# B&R Automation Studio project NAELD004C00R10L518F00 (part 36)

#### Act_Background.st
```iecst
(** 2020-05-26 **)
ACTION Act_Background:

	//Update Parameter
	IF bModuleOK = TRUE THEN

		tyParamInMove.diPosInUM		:= p_diMovePosInUM;
		tyParamInMove.diDistInUM	:= p_diMoveDistInUM;
		tyParamInMove.diVelInUMPS	:= p_diMoveVelInUMPS;
		tyParamInMove.diAcc			:= p_diMoveAcc;
		tyParamInMove.diDec			:= p_diMoveDec;

		fMotionCANUpdtDat(ADR(tyParamOut) , p_tyParamInConvert , tyParamOutDriver , tyParamInDriver , tyParamInMove , p_tyParamInHm , p_bDir, p_eNtParamMotorType);

		bWidthPosDiff	:= (tyParamOut.bIsHomed = FALSE) OR ((ABS((fAWWidthToPosInUM(p_diGoWidth , p_diWidthAtHmPos)) - tyParamOut.diActualPosInUM)) > 500);

		//p_tyParamInConvert.diPitchInUM	:= fPitchCalc(p_diWidthOffsetInUM , p_diMaxWidthInUM , p_diMinWidthInUM , p_diPitchInUM);

		fbFullMovAbsBl.tyParamInConvert					:= p_tyParamInConvert;

		IF p_bDir = TRUE THEN
			bOpenSen	:= tyParamOut.bFwdLmtSen;
			bCloseSen	:= tyParamOut.bRevLmtSen;
		ELSE
			bOpenSen	:= tyParamOut.bRevLmtSen;
			bCloseSen	:= tyParamOut.bFwdLmtSen;
		END_IF

		CASE p_eNtParamMotorType OF
			DeltaAsdaA2:
				CASE tyParamOut.udiAxisErrID OF
					8976:	sAxisErrTxt	:= 'Over Current';
					12560:	sAxisErrTxt	:= 'Over Voltage';
					12576:	sAxisErrTxt	:= 'Under Voltage';
					12592:	sAxisErrTxt	:= 'Input Power Phase Loss';
					12816:	sAxisErrTxt	:= 'Regeneration Error';
					12848:	sAxisErrTxt	:= 'Overload';
					12849:	sAxisErrTxt	:= 'Pre-overload Warning';
					13056:	sAxisErrTxt	:= 'U,V,W Wiring Error';
					16912:	sAxisErrTxt	:= 'IGBT Temperature Error';
					21296:	sAxisErrTxt	:= 'Memory Error';
					21569:	sAxisErrTxt	:= 'Emergency Stop Activated';
					21570:	sAxisErrTxt	:= 'Forward Limit Switch Error';
					21571:	sAxisErrTxt	:= 'Reverse Limit Switch Error';
					21572:	sAxisErrTxt	:= 'Forward Software Limit';
					21573:	sAxisErrTxt	:= 'Reverse Software Limit';
					21760:	sAxisErrTxt	:= 'DSP Firmware Upgrade';
					25088:	sAxisErrTxt	:= 'CANopen SYNC Error';
					25360:	sAxisErrTxt	:= 'CANopen Data Initial Error';
					25376:	sAxisErrTxt	:= 'Adjustment Error';
					28961:	sAxisErrTxt	:= 'Motor Protection Error';
					28962:	sAxisErrTxt	:= 'Motor Error';
					29445:	sAxisErrTxt	:= 'Encoder Error';
					29446:	sAxisErrTxt	:= 'Encoder Output Error';
					29968:	sAxisErrTxt	:= 'Serial Communication Error';
					29984:	sAxisErrTxt	:= 'Serial Communication Time Out';
					33024:	sAxisErrTxt	:= 'CANbus Error (Bus-off)';
					33040:	sAxisErrTxt	:= 'CANopen SDO receive buffer overrun';
					33056:	sAxisErrTxt	:= 'CANbus Error (Warning)';
					33072:	sAxisErrTxt	:= 'Node Guarding or Heartbeat Error';
					33280:	sAxisErrTxt	:= 'CANopen PDO Object Error';
					33792:	sAxisErrTxt	:= 'Over Speed';
					34304:	sAxisErrTxt	:= 'Abnormal Pulse Control Command';
					34320:	sAxisErrTxt	:= 'Full Closed Loop Excessive Deviation';
					34321:	sAxisErrTxt	:= 'Excessive Deviation';
				END_CASE

			SchneiderLexium28:
				CASE tyParamOut.udiAxisErrID OF
					8724:	sAxisErrTxt	:= 'Over Current';
					8976:	sAxisErrTxt	:= 'Motor Overload';
					8977:	sAxisErrTxt	:= 'Drive overload (foldback)';
					9088:	sAxisErrTxt	:= 'Calculated offsets for current sensors out OF range';
					9089:	sAxisErrTxt := 'Motor phase missing';
					9090:	sAxisErrTxt := 'Overcurrent detected at one OF the digital outputs';
					12560:	sAxisErrTxt	:= 'DC Bus Over Voltage';
					12576:	sAxisErrTxt	:= 'DC Bus Under Voltage';
					12672:	sAxisErrTxt	:= 'Braking Resistor Overload';
					12673:	sAxisErrTxt	:= 'Safety function Safe Torque Off (STO) triggered';
					12674:	sAxisErrTxt	:= 'DC bus voltage measurement';
					12675:	sAxisErrTxt	:= 'Missing mains supply, undervoltage mains supply';
					12676:	sAxisErrTxt := 'The encoder supply voltage has dropped under operational value';
					12677:	sAxisErrTxt := 'The multi turn encoder battery voltage has dropped under 3 Vdc';
					12678:	sAxisErrTxt := 'Internal position sync error detected.';
					12679:	sAxisErrTxt := 'Generic error code of the multi turn module is detected';
					12697:	sAxisErrTxt := 'Braking resistor overload';
					16512:	sAxisErrTxt	:= 'Drive overtemperature (IPM)';
					16513:	sAxisErrTxt	:= 'Drive overtemperature (controller)';
					16534:	sAxisErrTxt := 'Temperature sensor inoperative';
					17168:	sAxisErrTxt	:= 'Power stage overtemperature';
					17280:	sAxisErrTxt := 'The encoder temperature is too high';
					17424:	sAxisErrTxt	:= 'Motor overtemperature';
					21808:	sAxisErrTxt	:= 'System error detected (nonvolatilememory)';
					21893:	sAxisErrTxt	:= 'Error detected in non-volatile memory';
					21889:	sAxisErrTxt	:= 'System error detected (nonvolatile memory)';
					21890:	sAxisErrTxt	:= 'System error detected (CAN power supply)';
					21891:	sAxisErrTxt	:= 'System error detected (selftest)';
					21894:	sAxisErrTxt	:= 'System error detected (NV ACCESS)';
					25472:	sAxisErrTxt	:= 'Target position rejected';
					25985:	sAxisErrTxt	:= 'System error detected(FPGA)';
					28816:	sAxisErrTxt	:= 'System error detected (FPGA does NOT match firmware)';
					28817:	sAxisErrTxt	:= 'Emergency Stop Activated';
					28961:	sAxisErrTxt := 'Motor blocked';
					29080:	sAxisErrTxt := 'Commutation error detected';
					29568:  sAxisErrTxt	:= 'Error detected in communication with motor encoder';
					29574:	sAxisErrTxt	:= 'Drive is not synchronous wit master cycle';
					29581:	sAxisErrTxt := 'System error detected (encoder)';
					29587:	sAxisErrTxt	:= 'Encoder overvoltage or overcurrent';
					29592:	sAxisErrTxt := 'The returned position value are no longer considered valid';
					29593:	sAxisErrTxt := 'The multi turn encoder requires an explicit configuration command';
					30081:	sAxisErrTxt := 'Target position rejected';
					30082:	sAxisErrTxt := 'No target values received via the fieldbus';
					33072:	sAxisErrTxt	:= 'CANopen: Heartbeat error detected';
					33296:	sAxisErrTxt := 'R_PDO is too short';
					33921:	sAxisErrTxt	:= 'Actual Motor Velocity Too High';
					33553:	sAxisErrTxt	:= 'Motor torque too high FOR an excessive period OF time';
					33664:	sAxisErrTxt := 'Unstable current loop';
					33922:	sAxisErrTxt := 'Velocity deviation too high';
					34321:	sAxisErrTxt	:= 'Position deviation too high';
					34432:	sAxisErrTxt := 'Position deviation via signal output function MC_OK';
					34441:	sAxisErrTxt := 'Position deviation too high (following error)';
					61568:	sAxisErrTxt	:= 'Fieldbus: Communication	error detected';
					65282:	sAxisErrTxt	:= 'Not possible to read data of electronic motor nameplate';
					65296:	sAxisErrTxt	:= 'Forward Limit Switch Error';
					65297:	sAxisErrTxt	:= 'Reverse Limit Switch Error';
					65281:	sAxisErrTxt := 'System error detected';
					65298:	sAxisErrTxt	:= 'Forward Software Limit';
					65299:	sAxisErrTxt	:= 'Reverse Software Limit';
					65301:	sAxisErrTxt := 'The encoder firmware cannot operate on the provided hardware';

				END_CASE

			EstunPronet:
				CASE tyParamOut.udiAxisErrID OF
					65281:	sAxisErrTxt	:= 'Parameter breakdown';//A01
					65282:	sAxisErrTxt	:= 'AD shift channels breakdown';
					65283:	sAxisErrTxt	:= 'Overspeed';
					65284:	sAxisErrTxt	:= 'Overload';
					65285:	sAxisErrTxt := 'Position error counteroverflow ';
					65286:	sAxisErrTxt := 'Position error pulse overflow';
					65287:	sAxisErrTxt	:= 'The setting of electronic gear or given pulse frequency is not reasonable';
					65288:	sAxisErrTxt	:= 'The 1st channel of current detection is wrong.';
					65289:	sAxisErrTxt	:= 'The 2nd channel of current detection is wrong.';
					65290:	sAxisErrTxt	:= 'Incremental Encoder is break off.';//A10
					65292:	sAxisErrTxt	:= 'Overcurrent';
					65293:	sAxisErrTxt	:= 'Overvoltage';
					65294:	sAxisErrTxt	:= 'Undervoltage';
					65295:	sAxisErrTxt := 'Bleeder resistor error';
					65296:	sAxisErrTxt := 'Regeneration error';
					65297:	sAxisErrTxt := 'Resolver error';
					65298:	sAxisErrTxt := 'IGBT superheat alarm';
					65299:	sAxisErrTxt := 'Motor overheat alarm';
					65300:	sAxisErrTxt := 'Power line phase shortage';//A20
					65301:	sAxisErrTxt	:= 'Instantaneous power off alarm';
					65302:	sAxisErrTxt	:= 'Motor temperature detection sensor is break off.';
					65303:	sAxisErrTxt := 'Brake overcurrent alarm';//A23
					65305:	sAxisErrTxt := 'Motor power line U overcurrent';//A25
					65306:	sAxisErrTxt := 'Motor power line V overcurrent';//A26
					65307:	sAxisErrTxt := 'Motor power line W overcurrent';//A27
					65322:	sAxisErrTxt	:= 'Servomotor type error';//A42
					65323:	sAxisErrTxt	:= 'Servo drive type error';
					65325:	sAxisErrTxt	:= 'Absolute encoder multiturn information error';
					65326:	sAxisErrTxt	:= 'Absolute encoder multiturn information overflow';
					65327:	sAxisErrTxt	:= 'Battery voltage below 2.5V';
					65328:	sAxisErrTxt	:= 'Battery voltage below 3.1V';//A48
					65330:	sAxisErrTxt := 'Serial encoder communication overtime ';//A50
					65331:	sAxisErrTxt := 'Absolute encoder overspeed alarm detected';
					65332:  sAxisErrTxt	:= 'Absolute state of serial encoder error';
					65333:	sAxisErrTxt	:= 'Serial encoder calcaution error';
					65334:	sAxisErrTxt := 'Parity bit or end bit in serial encoder control domain error';
					65335:	sAxisErrTxt	:= 'Serial encoder communication data checking error';
					65336:	sAxisErrTxt := 'End bit in serial encoder control domain error';
					65338:	sAxisErrTxt := 'Serial encoder data empty';
					65339:	sAxisErrTxt := 'Serial encoder data format error';
					65340:	sAxisErrTxt := 'Communication module not detected ';//A60
					65341:	sAxisErrTxt := 'Communication unsuccessful';
					65342:	sAxisErrTxt := 'Servo drive can not receive the period data of communication module ';
					65343:	sAxisErrTxt := 'Communication module can not receive the servo drive response data.';
					65344:	sAxisErrTxt := 'Communication module and bus connectionless';
					65346:	sAxisErrTxt := 'CAN communication abnormal';
					65347:	sAxisErrTxt := 'Receiving heartbeat timeout';
					65349:	sAxisErrTxt := 'Synchronization signal monitoring cycle is longer than setting';
					65362: sAxisErrTxt	:= 'Torque output alarm';
				END_CASE
		END_CASE

	ELSE

		tyParamOut.bAxisErr			:= FALSE;
		tyParamOut.bFwdLmtSen		:= FALSE;
		tyParamOut.bInPos			:= FALSE;
		tyParamOut.bIsHomed			:= FALSE;
		tyParamOut.bPosDiff			:= TRUE;
		tyParamOut.bPwrOn			:= FALSE;
		tyParamOut.bRevLmtSen		:= FALSE;
		tyParamOut.bStopped			:= TRUE;
		tyParamOut.diActualPosInUM	:= 0;
		tyParamOut.diHmAcc			:= 0;
		tyParamOut.diHmSpdForSwitch	:= 0;
		tyParamOut.diHmSpdForZero	:= 0;
		tyParamOut.diProfileAcc		:= 0;
		tyParamOut.diProfileDec		:= 0;
		tyParamOut.udiAxisErrID		:= 0;

		bWidthPosDiff				:= TRUE;

	END_IF

	//Abnormal Movement
//	IF eStatus1 <> Error THEN
//		IF p_bOps = TRUE AND eStatus = Idle THEN
//			IF (ABS(tyParamOut.diActualPosInUM - diActualPosInUMOld) > 2000) AND (ABS(tyParamOut.diActualPosInUM - diActualPosInUMOld) < 10000) THEN
//				eStatus1	:= Error;
//				udiStatus1	:= 10000;	//Axis Move Abnormally By External Force
//
//				fMotionCANRstCtrlWord(ADR(tyParamOutDriver));
//				p_eAct	:= PPActIdle;
//				eStat	:= PPActIdle;
//			END_IF
//		ELSE
//			diActualPosInUMOld	:= tyParamOut.diActualPosInUM;
//		END_IF
//	END_IF

	//Reset Error
	IF (eStatus1 = Error) AND bRstErr THEN
		eStatus1	:= Idle;
		udiStatus1	:= 0;
	END_IF

	//Request Position To Movement Out Of Range
	IF p_bOps
		AND((tyParamInMove.diPosInUM < p_diMinAbsPosInUM) OR (tyParamInMove.diPosInUM > p_diMaxAbsPosInUM))
		AND (eStatus2 <> Error) THEN
		eStatus2	:= Error;
		udiStatus2	:= 10029;	//Request Absolute Position Out Of Range

		fMotionCANRstCtrlWord(ADR(tyParamOutDriver));
		p_eAct	:= PPActIdle;
		eStat	:= PPActIdle;
	END_IF

	//Reset Error
	IF (eStatus2 = Error) AND bRstErr THEN
		eStatus2	:= Idle;
		udiStatus2	:= 0;
	END_IF

	//Sensor Interrupt
	IF (bNotInterruptible = TRUE OR bJogging) AND eStatus3 <> Error THEN

		IF p_bInletSensor = TRUE THEN
			eStatus3	:= Error;
			udiStatus3	:= 10030;	//Inlet Sensor Interrupt Auto Width Movement

			fMotionCANRstCtrlWord(ADR(tyParamOutDriver));
			p_eAct	:= PPActIdle;
			eStat	:= PPActIdle;

		ELSIF p_bOutletSensor = TRUE THEN
			eStatus3	:= Error;
			udiStatus3	:= 10031;	//Outlet Sensor Interrupt Auto Width Movement

			fMotionCANRstCtrlWord(ADR(tyParamOutDriver));
			p_eAct	:= PPActIdle;
			eStat	:= PPActIdle;

		ELSIF p_bClearSensor = TRUE THEN
			eStatus3	:= Error;
			udiStatus3	:= 10032;	//Clear Sensor Interrupt Auto Width Movement

			fMotionCANRstCtrlWord(ADR(tyParamOutDriver));
			p_eAct	:= PPActIdle;
			eStat	:= PPActIdle;

		ELSIF p_bMiddleSensor = TRUE THEN
			eStatus3	:= Error;
			udiStatus3	:= 10033;	//Middle Sensor Interrupt Auto Width Movement

			fMotionCANRstCtrlWord(ADR(tyParamOutDriver));
			p_eAct	:= PPActIdle;
			eStat	:= PPActIdle;

		ELSIF p_bInterruptSensor = TRUE THEN
			eStatus3	:= Error;
			udiStatus3	:= 10034;	//Sensor Interrupt Auto Width Movement

			fMotionCANRstCtrlWord(ADR(tyParamOutDriver));
			p_eAct	:= PPActIdle;
			eStat	:= PPActIdle;

		ELSIF p_bCloseInterruptSensor = TRUE AND bJogOpen = FALSE THEN
			eStatus3	:= Error;
			udiStatus3	:= 10047;	//Sensor Interrupt Auto Width Movement

			fMotionCANRstCtrlWord(ADR(tyParamOutDriver));
			p_eAct	:= PPActIdle;
			eStat	:= PPActIdle;

		ELSIF p_bOpenInterruptSensor = TRUE AND bJogClose = FALSE THEN
			eStatus3	:= Error;
			udiStatus3	:= 10048;	//Sensor Interrupt Auto Width Movement

			fMotionCANRstCtrlWord(ADR(tyParamOutDriver));
			p_eAct	:= PPActIdle;
			eStat	:= PPActIdle;
		END_IF

	END_IF

	//Reset Error
	IF (eStatus3 = Error AND bRstErr)
		OR (p_bOpenInterruptSensor AND eStat = PPActJogClose)
		OR (p_bCloseInterruptSensor AND eStat = PPActJogOpen)
		THEN
		eStatus3	:= Idle;
		udiStatus3	:= 0;
	END_IF

	IF bRstErr THEN
		udiStatus	:= 0;
		bJogging	:= FALSE;
		bJogClose	:= FALSE;
		bJogOpen	:= FALSE;
	END_IF

	fbServoModuleOk(IN:= bModuleOK);
	fbServoModuleNotOk(IN:= bModuleOK = FALSE);
	IF fbServoModuleNotOk.Q AND udiStatus <> 10001 THEN

		bModuleNotOK		:= TRUE;
		bModuleNotOKLock	:= TRUE;
		usiRstStep	:= 0;
		tyParamOutDriver.uiCtrlword_6040	:= 0;
		tyParamOutDriver.siModOfOpt_6060	:= 0;
		tyParamOutDriver.diTargetPos_607A	:= 0;
		tyParamOutDriver.udiMoveSpd_6081	:= 0;
		tyParamOutDriver.siHmMethod_6098	:= 0;
		tyParamOutDriver.diJogVel_60FF		:= 0;

		CASE p_eNtParamMotorType OF

			DeltaAsdaA2:
				fbModuleOK(bModuleOK:= FALSE);
				IF eStatus = Idle THEN
					eAct	:= PPActRstNode;
				END_IF

				IF (eStatus = Done OR eStatus = Error)AND eStat = PPActRstNode THEN

					eAct	:= PPActIdle;
				END_IF

			EstunPronet:
				fbModuleOK(bModuleOK:= FALSE);
				IF eStatus = Idle THEN
					eAct	:= PPActRstNode;
				END_IF

				IF (eStatus = Done OR eStatus = Error)AND eStat = PPActRstNode THEN

					eAct	:= PPActIdle;
				END_IF

			SchneiderLexium28:
			// Do Nothing
		END_CASE

	ELSIF bModuleNotOK = TRUE AND fbServoModuleOk.Q THEN

		CASE usiRstStep OF

			0:
				IF eStatus = Idle THEN
					eAct	:= PPActRstAxisErr;
				END_IF

				IF eStatus = Done AND eStat = PPActRstAxisErr THEN
					eAct	:= PPActIdle;
					usiRstStep	:= 4;
				END_IF

			4: tyParamOutDriver.siModOfOpt_6060 := 1;
				usiRstStep	:= 5;

			5: tyParamOutDriver.siModOfOpt_6060 := 1;
				fbRstNodeTimer(IN:=TRUE);

				IF tyParamInDriver.siModOfOptDisp_6061 = 1 THEN
					usiRstStep	:= 6;
					fbRstNodeTimer(IN:=FALSE);
				ELSIF fbRstNodeTimer.Q THEN
					usiRstStep	:= 8;
					fbRstNodeTimer(IN:=FALSE);
				END_IF

			6: tyParamOutDriver.siModOfOpt_6060 := 6;
				fbRstNodeTimer(IN:=FALSE);
				usiRstStep	:= 7;

			7: tyParamOutDriver.siModOfOpt_6060 := 6;
				fbRstNodeTimer(IN:=TRUE);

				IF tyParamInDriver.siModOfOptDisp_6061 = 6 THEN
					usiRstStep	:= 10;
					fbRstNodeTimer(IN:=FALSE);
				ELSIF fbRstNodeTimer.Q THEN
					usiRstStep	:= 9;
					fbRstNodeTimer(IN:=FALSE);
				END_IF

			8:	fbModuleOK(bEn := TRUE, bModuleOK:= FALSE);
				fbRstNodeTimer(IN:=FALSE);
				usiRstStep	:= 9;

			9:	fbModuleOK(bModuleOK:= FALSE);
				IF eStatus = Idle THEN
					eAct	:=PPActRstNode;
				END_IF

				IF eStatus = Done AND eStat = PPActRstNode THEN
					usiRstStep	:= 0;
					eAct		:= PPActIdle;
				END_IF

			10:IF eStatus = Idle THEN
					eAct	:= PPActRstAxisErr;
				END_IF

				IF eStatus = Done AND eStat = PPActRstAxisErr THEN
					eAct			:=PPActIdle;
					usiRstStep	:= 11;
				END_IF

			11:

				IF eStatus = Idle THEN
					eAct	:= PPActSDOWrite;
				END_IF

				IF eStatus = Done AND eStat = PPActSDOWrite THEN
					eAct			:= PPActIdle;
					usiRstStep	:= 13;

				ELSIF udiStatus = 10028 THEN
					eAct			:= PPActIdle;
					usiRstStep	:= 13;
				END_IF

			13: bModuleNotOK	:= FALSE;
				usiRstStep	:= 0;
		END_CASE
	ELSE
		eAct	:= PPActIdle;

	END_IF

	IF tyParamOut.bPosDiff = FALSE THEN
		tyParamOutDriver.uiCtrlword_6040.4	:= FALSE;
	END_IF

END_ACTION
```

#### Act_InitGlobal.st
```iecst
(** 2019-04-09 **)
ACTION Act_InitGlobal:

	(* Always Change If Project Change *)

	//Pass Data To Link
	p_bLinkOpsRun ACCESS p_OpsRun;
	p_bLinkStartupRun ACCESS p_StartupRun;
	p_bLinkPullConvPullerExtCtrl ACCESS p_PullConvPullerExtCtrl;
	p_bLinkPullConvPullerRetCtrl ACCESS p_PullConvPullerRetCtrl;
	p_bLinkDIPullerExtRS ACCESS p_DIPullerExtRS;
	p_bLinkDIPullerRetRS ACCESS p_DIPullerRetRS;
	p_bLinkDIPullerExtSlwRS ACCESS p_DIPullerExtSlwSen;
	p_bLinkDIPullerRetSlwRS ACCESS p_DIPullerRetSlwSen;
	p_dintLinkPullerRetSpd ACCESS p_ProdRcpCurrRcp1MtrPshrExtSpd;
	p_dintLinkPullerRetTrq ACCESS p_ProdRcpCurrRcp1MtrPshrExtTorq;
	p_bLinkDIPullerRotHmRS ACCESS p_DIPullerRotHmRS;

	p_diLinkMag1TravPos ACCESS p_MagRcpCurrRcpMag1TravPos;
	p_diLinkMag2TravPos ACCESS p_MagRcpCurrRcpMag2TravPos;
	p_diLinkMag3TravPos ACCESS p_MagRcpCurrRcpMag3TravPos;
	p_diLinkTravActualPos ACCESS p_TravActualPos;
	p_bProjCurtainSenPrep ACCESS p_NtParamProjCurtainSenPrep; //shutter become individual : interrupt sensor
	p_diRcp1MtrPshrExtTorq ACCESS p_ProdRcpCurrRcp1MtrPshrExtTorq;
	p_bMagWidthChkSen ACCESS p_DIMagWidthChkSen;
	p_tyLinkTorqParam ACCESS p_NtParamPPTorqParam;

	//Pass Data To Internal Use
	p_udiRstErr ACCESS p_RstErrReset;
	p_bEn ACCESS p_DISimServoEn;
	p_bPrep ACCESS p_NtParamProjServoPullPusherPrep;
	p_bOps ACCESS p_OpsStatusRun;
	p_bManual ACCESS p_UIMnlMod;
	p_tyTuning ACCESS p_NtParamPPTuning;
//	p_diJogVelInUMPS ACCESS p_UIMnlPPJogSpd;
	p_diMovePosInUM ACCESS p_UIMnlPPTargetPos;
	p_diMoveDistInUM ACCESS p_UIMnlPPStepSize;
	p_diMoveVelInUMPS ACCESS p_NtParamPPAutoSpd;
	p_diMoveAcc ACCESS p_NtParamPPAcc;
	p_diMoveDec ACCESS p_NtParamPPDec;
	p_diWidthOffsetInUM ACCESS p_NtParamWidthOffset;
	p_bDir ACCESS p_NtParamPPDir;
	p_bDirBl ACCESS p_NtParamPPDirBl;
	p_usiNode ACCESS p_NtParamPPNode;
	p_sDevice ACCESS p_NtParamPPDevice;
	p_sProgNm ACCESS p_NtParamPPProgNm;
	p_diMoveBacklashDistInUM ACCESS p_NtParamPPMovBlDistInUM;
	p_diPitchInUM ACCESS p_NtParamPPPitchInUM;
	p_tyParamInHm ACCESS p_NtParamPPParamInHm;
	p_tyParamInConvert ACCESS p_NtParamPPParamInConvert;
	p_bNtSettingsLoadDone ACCESS p_StartupNtSettingsLoadDone;
	p_eNtParamMotorType ACCESS p_NtParamPPMotorType;

	p_bInletShutterCloseRS ACCESS p_DIInShutterCloseRS;
	p_bOutletShutterCloseRS ACCESS p_DIOutShutterCloseRS;
	p_bProjInletShutPrep ACCESS p_NtParamProjInletShutPrep;
	p_bProjOutletShutPrep ACCESS p_NtParamProjOutletShutPrep;

	p_bInletShutterCloseRS2 ACCESS p_DIInShutterCloseRS2;
	p_bInletShutterCloseRS3 ACCESS p_DIInShutterCloseRS3;

	(* Always Change If Project Change *)

END_ACTION
```

#### Act_Initial.st
```iecst
(** 2020-03-16 **)
ACTION Act_Initial:

	//Initial
	sStatTxt	:= a_sStatText[eStat];

	tyParamInMove.diBacklashDistInUM	:= p_diMoveBacklashDistInUM;
	tyParamInMove.diAcc					:= p_diMoveAcc;
	tyParamInMove.diDec					:= p_diMoveDec;

	//p_tyParamInConvert.diPitchInUM	:= fPitchCalc(p_diWidthOffsetInUM , p_diMaxWidthInUM , p_diMinWidthInUM , p_diPitchInUM);

	fbModuleOK.sDevice	:= p_sDevice;
	fbModuleOK.usiNode	:= p_usiNode;
	fbModuleOK.tDlyTm	:= T#5s;
	fbModuleOK(bEn := FALSE);

	fbSDOWrite.sDevice	:= p_sDevice;
	fbSDOWrite.usiNode	:= p_usiNode;
	fbSDOWrite.eMotorType	:= p_eNtParamMotorType;
	fbSDOWrite(bEn := FALSE);

	fbFullMovAbsBl.p_tyParamOutDriver				:= ADR(tyParamOutDriver);
	fbFullMovAbsBl.tyParamInMove.diBacklashDistInUM	:= p_diMoveBacklashDistInUM;
	fbFullMovAbsBl.tyParamInMove.diAcc				:= p_diMoveAcc;
	fbFullMovAbsBl.tyParamInMove.diDec				:= p_diMoveDec;
	//fbFullMovAbsBl.tyParamInConvert					:= p_tyParamInConvert;
	fbFullMovAbsBl.bDir								:= p_bDir;
	fbFullMovAbsBl.bDirBl							:= p_bDirBl;
	fbFullMovAbsBl.bNoIndexPulse					:= p_bNoIndexPulse;
	fbFullMovAbsBl.eMotorType						:= p_eNtParamMotorType;
	fbFullMovAbsBl(bEn := FALSE);

	fbFullMovAbs.p_tyParamOutDriver					:= ADR(tyParamOutDriver);
	fbFullMovAbs.tyParamInMove.diBacklashDistInUM	:= p_diMoveBacklashDistInUM;
	fbFullMovAbs.tyParamInMove.diAcc				:= p_diMoveAcc;
	fbFullMovAbs.tyParamInMove.diDec				:= p_diMoveDec;
	fbFullMovAbs.tyParamInConvert					:= p_tyParamInConvert;
	fbFullMovAbs.bDir								:= p_bDir;
	fbFullMovAbs.bNoIndexPulse						:= p_bNoIndexPulse;
	fbFullMovAbs.eMotorType							:= p_eNtParamMotorType;
	fbFullMovAbs(bEn := FALSE);

	fbFullHm.p_tyParamOutDriver	:= ADR(tyParamOutDriver);
	fbFullHm.bDir				:= p_bDir;
	fbFullHm.bNoIndexPulse		:= p_bNoIndexPulse;
	fbFullHm.eMotorType			:= p_eNtParamMotorType;
	fbFullHm(bEn := FALSE);

	fbPwrOn.p_tyParamOutDriver	:= ADR(tyParamOutDriver);
	fbPwrOn.eMotorType			:= p_eNtParamMotorType;
	fbPwrOn(bEn := FALSE);

	fbPwrOff.p_tyParamOutDriver	:= ADR(tyParamOutDriver);
	fbPwrOff.eMotorType			:= p_eNtParamMotorType;
	fbPwrOff(bEn := FALSE);

	fbHoming.p_tyParamOutDriver	:= ADR(tyParamOutDriver);
	fbHoming.bDir				:= p_bDir;
	fbHoming.bNoIndexPulse		:= p_bNoIndexPulse;
	fbHoming.eMotorType			:= p_eNtParamMotorType;
	fbHoming(bEn := FALSE);

	fbMovAbs.p_tyParamOutDriver					:= ADR(tyParamOutDriver);
	fbMovAbs.tyParamInMove.diBacklashDistInUM	:= p_diMoveBacklashDistInUM;
	fbMovAbs.tyParamInMove.diAcc				:= p_diMoveAcc;
	fbMovAbs.tyParamInMove.diDec				:= p_diMoveDec;
	fbMovAbs.tyParamInConvert					:= p_tyParamInConvert;
	fbMovAbs.bDir								:= p_bDir;
	fbMovAbs.eMotorType							:= p_eNtParamMotorType;
	fbMovAbs(bEn := FALSE);

	fbMovRel.p_tyParamOutDriver					:= ADR(tyParamOutDriver);
	fbMovRel.tyParamInMove.diBacklashDistInUM	:= p_diMoveBacklashDistInUM;
	fbMovRel.tyParamInMove.diAcc				:= p_diMoveAcc;
	fbMovRel.tyParamInMove.diDec				:= p_diMoveDec;
	fbMovRel.tyParamInConvert					:= p_tyParamInConvert;
	fbMovRel.bDir								:= p_bDir;
	fbMovRel.eMotorType							:= p_eNtParamMotorType;
	fbMovRel(bEn := FALSE);

	fbJog.p_tyParamOutDriver	:= ADR(tyParamOutDriver);
	fbJog.tyParamInConvert		:= p_tyParamInConvert;
	fbJog.eMotorType			:= p_eNtParamMotorType;
	fbJog(bEn := FALSE);

	fbRstAxisErr.p_tyParamOutDriver	:= ADR(tyParamOutDriver);
	fbRstAxisErr(bEn := FALSE);

	fbStop.p_tyParamOutDriver	:= ADR(tyParamOutDriver);
	fbStop(bEn := FALSE);

	fbSDOWriteTorque.pDevice := ADR(p_sDevice);
	fbSDOWriteTorque.node	 := p_usiNode;

	fbSDOWriteTorque.index	:= 16#210C;
	fbSDOWriteTorque.subindex	:= 0;
	fbSDOWriteTorque.datalen	:= 2;

	bModuleNotOK	:= TRUE;

END_ACTION
```

#### Act_InitLocal.st
```iecst
(** 2020-05-26 **)
ACTION Act_InitLocal:

	//Input Reference Link To Local Variable
	p_eAct ACCESS ADR(eAct);
	p_udiRstErr ACCESS ADR(udiRstErr);
	p_bPrep ACCESS ADR(bPrep);
	p_bEn ACCESS ADR(bEn);
	p_bDis ACCESS ADR(bDis);
	p_bOps ACCESS ADR(bOps);
	p_bManual ACCESS ADR(bManual);
	p_diWidthAtHmPos ACCESS ADR(diWidthAtHmPos);
	p_tyTuning ACCESS ADR(tyTuning);
	p_diGoWidth ACCESS ADR(diGoWidth);
	p_diJogVelInUMPS ACCESS ADR(diJogVelInUMPS);
	p_diMovePosInUM ACCESS ADR(diMovePosInUM);
	p_diMoveDistInUM ACCESS ADR(diMoveDistInUM);
	p_diMoveVelInUMPS ACCESS ADR(diMoveVelInUMPS);
	p_diMoveAcc ACCESS ADR(diMoveAcc);
	p_diMoveDec ACCESS ADR(diMoveDec);
	p_diMinAbsPosInUM ACCESS ADR(diMinAbsPosInUM);
	p_diMaxAbsPosInUM ACCESS ADR(diMaxAbsPosInUM);
	p_diMinWidthInUM ACCESS ADR(diMinWidthInUM);
	p_diMaxWidthInUM ACCESS ADR(diMaxWidthInUM);
	p_diWidthOffsetInUM ACCESS ADR(diWidthOffsetInUM);
	p_bInletSensor ACCESS ADR(bInletSensor);
	p_bOutletSensor ACCESS ADR(bOutletSensor);
	p_bClearSensor ACCESS ADR(bClearSensor);
	p_bMiddleSensor ACCESS ADR(bMiddleSensor);
	p_bInterruptSensor ACCESS ADR(bInterruptSensor);
	p_bOpenInterruptSensor ACCESS ADR(bOpenInterruptSensor);
	p_bCloseInterruptSensor ACCESS ADR(bCloseInterruptSensor);
	p_bDir ACCESS ADR(bDir);
	p_bDirBl ACCESS ADR(bDirBl);
	p_bNoIndexPulse ACCESS ADR(bNoIndexPulse);
	p_usiNode ACCESS ADR(usiNode);
	p_sDevice ACCESS ADR(sDevice);
	p_sProgNm ACCESS ADR(sProgNm);
	p_diMoveBacklashDistInUM ACCESS ADR(diMoveBacklashDistInUM);
	p_diPitchInUM ACCESS ADR(diPitchInUM);
	p_tyParamInHm ACCESS ADR(tyParamInHm);
	p_tyParamInConvert ACCESS ADR(tyParamInConvert);
	p_bNtSettingsLoadDone ACCESS ADR(bNtSettingsLoadDone);
	p_eNtParamMotorType ACCESS ADR(eMotorType);
	p_diServoTorque ACCESS ADR(diServoTorque);
	p_diRcp1MtrPshrExtTorq ACCESS ADR(diRcp1MtrPshrExtTorq);
END_ACTION
```

#### Act_Link.st
```iecst
(** 2019-03-29 **)
ACTION Act_Link:
	diRcp1MtrPshrExtTorq	 := p_tyLinkTorqParam.usiStartTorque + (((p_diRcp1MtrPshrExtTorq -10)/10)*p_tyLinkTorqParam.uiRatio/100);//15~30N , Rcp1 torque

	IF p_bProjInletShutPrep = TRUE THEN

		IF p_bProjCurtainSenPrep = FALSE THEN //standard
			IF p_bInletShutterCloseRS
				THEN
				bInterruptSensor1 := TRUE;
			ELSE
				bInterruptSensor1 := FALSE;
			END_IF
		ELSE
			IF eStat <> PPActJogClose THEN
				IF ABS(p_diLinkMag1TravPos - p_diLinkTravActualPos) < 500 THEN
					bInterruptSensor1 := p_bInletShutterCloseRS;
				ELSIF ABS(p_diLinkMag2TravPos - p_diLinkTravActualPos) < 500 THEN
					bInterruptSensor1 := p_bInletShutterCloseRS2;
				ELSIF ABS(p_diLinkMag3TravPos - p_diLinkTravActualPos) < 500 THEN
					bInterruptSensor1 := p_bInletShutterCloseRS3;
				END_IF
			END_IF
		END_IF
	ELSE
		bInterruptSensor1 := FALSE;
	END_IF

//	IF p_bProjOutletShutPrep = TRUE THEN
//		IF p_bOutletShutterCloseRS
//			THEN
//			bInterruptSensor2 := TRUE;
//		ELSE
//			bInterruptSensor2 := FALSE;
//		END_IF
//	ELSE
//		bInterruptSensor2 := FALSE;
//	END_IF

//	IF (usiJogFwdStep = 40 AND p_eAct = PPActJogOpen) OR (usiJogRevStep = 40 AND p_eAct = PPActJogClose) THEN
//		bInterruptSensor3	:= NOT p_bMagWidthChkSen;
//	END_IF
//	IF p_eAct = PPActIdle OR p_eAct = PPActStop THEN
//		bInterruptSensor3  := FALSE;
//	END_IF

	p_bInterruptSensor := bInterruptSensor3 OR bInterruptSensor2 OR bInterruptSensor1;// OR p_bLinkSafetyRelay = FALSE;

END_ACTION
```

#### Act_LinkAction.st
```iecst
(** 2019-10-21 **)
ACTION Act_LinkAction:

	IF bModuleNotOK THEN
		p_eAct ACCESS ADR(eAct);
	ELSE
		IF p_bLinkStartupRun = TRUE THEN
			p_eAct ACCESS p_StartupServoPPAct;
		ELSIF p_bLinkOpsRun = TRUE OR p_bManual = TRUE THEN
			IF p_bLinkPullConvPullerExtCtrl AND NOT bJogFwdDone
				//AND NOT p_bLinkDIPullerExtRS
				THEN
				bJogStopDone := FALSE;

				CASE usiJogFwdStep OF

					0:
						memcpy(ADR(fbSDOWriteTorque.data0),ADR(udiMaxTorque),1);
						memcpy(ADR(fbSDOWriteTorque.data1),ADR(udiMaxTorque)+1,1);
						IF eStat <> PPActIdle THEN
							p_eAct := PPActIdle;
							usiJogFwdStep := 20;
						ELSE
							usiJogFwdStep := 20;
						END_IF

					20:
						fbSDOWriteTorque(enable := TRUE);
						IF fbSDOWriteTorque.status = 65535 THEN
							usiJogFwdStep := 22;
						END_IF

					22:
						fbSDOWriteTorque(enable := TRUE);
						IF fbSDOWriteTorque.status = 0 THEN
							fbSDOWriteTorque(enable := FALSE);
							usiJogFwdStep := 30;
						END_IF

					30:
						IF tyParamOut.bPwrOn = FALSE THEN
							p_eAct := PPActPwrOn;

							IF tyParamOut.bPwrOn THEN
								p_eAct := PPActIdle;
								usiJogFwdStep := 40;
							END_IF
						ELSE
							p_eAct := PPActIdle;
							usiJogFwdStep := 40;

						END_IF

					40:
						p_eAct := PPActJogOpen;

						IF EDGEPOS(p_bLinkDIPullerExtSlwRS) THEN
							bExtSlowSpd := TRUE;
							p_eAct := PPActIdle;
						END_IF

						IF p_bLinkDIPullerExtSlwRS OR p_bLinkDIPullerExtRS  THEN
							p_diJogVelInUMPS := diSlowSpeed;

						ELSE
							IF p_bManual THEN
								p_diJogVelInUMPS ACCESS p_UIMnlPPJogSpd;
							ELSE
									p_diJogVelInUMPS := udiJogSpdAuto; //325000;//290000;
							END_IF
						END_IF

					//	IF (eStat = PPActJogOpen AND eMainStatus = Done)
					//		OR p_bLinkDIPullerExtRS
						IF p_bLinkDIPullerExtRS
							THEN
							p_eAct := PPActIdle;
							p_diJogVelInUMPS := 0;
							usiJogFwdStep := 50;

						END_IF

					50:
						p_eAct := PPActJogStop;
						p_diJogVelInUMPS := 0;
						IF (eStat = PPActJogStop AND eMainStatus = Done)
							THEN
							p_eAct := PPActIdle;
							usiJogFwdStep := 0;
							bJogFwdDone := TRUE;
						END_IF

				END_CASE

			ELSIF p_bLinkPullConvPullerRetCtrl AND NOT bJogRevDone
				//AND NOT p_bLinkDIPullerRetRS
				THEN
				bJogStopDone := FALSE;
				CASE usiJogRevStep OF

					0:
						IF p_bManual THEN
							memcpy(ADR(fbSDOWriteTorque.data0),p_UIMnlMtrPshrRetTorq,1);
							memcpy(ADR(fbSDOWriteTorque.data1),p_UIMnlMtrPshrRetTorq+1,1);
						ELSE
							memcpy(ADR(fbSDOWriteTorque.data0),ADR(diRcp1MtrPshrExtTorq),1);
							memcpy(ADR(fbSDOWriteTorque.data1),ADR(diRcp1MtrPshrExtTorq)+1,1);
						END_IF
						IF eStat <> PPActIdle THEN
							p_eAct := PPActIdle;
							usiJogRevStep := 20;
						ELSE
							usiJogRevStep := 20;
						END_IF

					20:
						fbSDOWriteTorque(enable := TRUE);
						IF fbSDOWriteTorque.status = 65535 THEN
							usiJogRevStep := 22;
						END_IF

					22:
						fbSDOWriteTorque(enable := TRUE);
						IF fbSDOWriteTorque.status = 0 THEN
							fbSDOWriteTorque(enable := FALSE);
							usiJogRevStep := 30;
						END_IF

					30:
						IF tyParamOut.bPwrOn = FALSE THEN
							p_eAct := PPActPwrOn;
							IF tyParamOut.bPwrOn THEN
								p_eAct := PPActIdle;
								usiJogRevStep := 40;
							END_IF
						ELSE
							p_eAct := PPActIdle;
							usiJogRevStep := 40;

						END_IF

					40:
						p_eAct := PPActJogClose;

						IF EDGEPOS(p_bLinkDIPullerRetSlwRS) THEN
							p_eAct := PPActIdle;
						END_IF

						IF p_bLinkDIPullerRetSlwRS OR p_bLinkDIPullerRetRS THEN
							p_diJogVelInUMPS := diSlowSpeed;
						ELSE
							IF p_bManual THEN
								p_diJogVelInUMPS ACCESS p_UIMnlPPJogSpd;
							ELSE
								p_diJogVelInUMPS := p_dintLinkPullerRetSpd * uiJogSpdRatio; //40625//36250
							END_IF

						END_IF

					//	IF (eStat = PPActJogClose AND eMainStatus = Done)
					//		OR p_bLinkDIPullerRetRS
						IF p_bLinkDIPullerRetRS
							THEN
							p_eAct := PPActIdle;
							p_diJogVelInUMPS := 0;
							usiJogRevStep := 50;

						END_IF

					50:
						p_eAct := PPActJogStop;
						p_diJogVelInUMPS := 0;
						IF (eStat = PPActJogStop AND eMainStatus = Done)
						THEN
							p_eAct := PPActIdle;
							usiJogRevStep := 0;
							bJogRevDone := TRUE;
						END_IF

				END_CASE
			ELSE

				IF bJogStopDone = FALSE THEN
					p_eAct := PPActJogStop;
				END_IF

				usiJogFwdStep := 0;
				usiJogRevStep := 0;
				p_diJogVelInUMPS := 0;

				IF eStat = PPActJogStop AND eMainStatus = Done THEN
					p_eAct := PPActIdle;
					bJogStopDone := TRUE;
				END_IF

				IF tyParamInDriver.uiErrCode_603F <> 0 THEN //error 12592
					tyParamOutDriver.uiCtrlword_6040 := 0; //0111 (7)> 1111 (15)
				END_IF

			END_IF

		ELSE
			IF bRstAndExt = FALSE THEN
				p_eAct ACCESS ADR(eAct);
				usiJogFwdStep := 0;
				usiJogRevStep := 0;
				usiRstJogStep := 0;
				p_diJogVelInUMPS := 0;
				IF bModuleNotOK = FALSE THEN
					IF eStatus <> Idle THEN
						p_eAct := PPActIdle;
						IF eStat = PPActIdle AND eMainStatus = Done THEN
							p_eAct := PPActIdle;
						END_IF
					END_IF
				END_IF
			ELSIF p_bLinkDIPullerRetRS OR p_bLinkDIPullerRotHmRS THEN
				bRstAndExt := FALSE;

			ELSE //reset do extend
				p_eAct ACCESS ADR(eAct);
				CASE usiRstJogStep OF
					0:
						fbPwrOnDlyTmr(IN:=tyParamOut.bPwrOn = FALSE);
						IF tyParamOut.bPwrOn = FALSE AND fbPwrOnDlyTmr.Q THEN
							p_eAct := PPActPwrOn;

							IF tyParamOut.bPwrOn THEN
								fbPwrOnDlyTmr(IN:=FALSE);
								p_eAct := PPActIdle;
								usiRstJogStep := 1;
							END_IF
						ELSE
							fbPwrOnDlyTmr(IN:=FALSE);
							p_eAct := PPActIdle;
							usiRstJogStep := 1;

						END_IF
					1:
						p_eAct := PPActJogOpen;

						IF EDGEPOS(p_bLinkDIPullerExtSlwRS) THEN
							p_eAct := PPActIdle;
						END_IF

						IF p_bLinkDIPullerExtSlwRS OR p_bLinkDIPullerExtRS OR bExtSlowSpd THEN
							p_diJogVelInUMPS := diSlowSpeed;

						ELSE
							p_diJogVelInUMPS := 12000; //50%

						END_IF

						IF p_bLinkDIPullerExtRS	THEN
							p_eAct := PPActIdle;
							p_diJogVelInUMPS := 0;
							usiRstJogStep := 2;
							bTurnToHm	:= TRUE; // output
							bExtSlowSpd := FALSE;

						END_IF

					2:
						p_eAct := PPActJogStop;
						p_diJogVelInUMPS := 0;
						IF (eStat = PPActJogStop AND eMainStatus = Done)
							THEN
							p_eAct := PPActIdle;
							bRstAndExt := FALSE;
						END_IF
				END_CASE

			END_IF
		END_IF //end run/manual
	END_IF

	IF EDGENEG(p_bManual) OR EDGENEG(p_bLinkOpsRun) OR EDGENEG(p_bLinkStartupRun) THEN
		tyParamOutDriver.uiCtrlword_6040	:= 0;
	END_IF

	IF (eStat = PPActJogClose AND p_bLinkDIPullerRetRS)
		OR (eStat = PPActJogOpen AND p_bLinkDIPullerExtRS)
		THEN
		p_diJogVelInUMPS := 0;
	END_IF

	IF p_bLinkDIPullerRetRS = FALSE THEN
		bJogRevDone := FALSE;
	END_IF

	IF p_bLinkDIPullerExtRS = FALSE THEN
		bJogFwdDone := FALSE;
	END_IF

END_ACTION
```

#### Act_Main.st
```iecst
(** 2020-05-26 **)
ACTION Act_Main:

	//Main
IF bModuleNotOK = FALSE THEN

		CASE eStat OF

			PPActIdle:
				IF eStatus <> Idle THEN	//Reset Data
					//Private
					fbStop(bEn := FALSE);
					fbRstAxisErr(bEn := FALSE);
					fbJog(bEn := FALSE);
					fbMovRel(bEn := FALSE);
					fbMovAbs(bEn := FALSE);
					fbHoming(bEn := FALSE);
					fbPwrOff(bEn := FALSE);
					fbPwrOn(bEn := FALSE);
					fbFullHm(bEn := FALSE);
					fbFullMovAbs(bEn := FALSE);
					fbFullMovAbsBl(bEn := FALSE);
					fbSDOWrite(bEn := FALSE);
					fbTm(IN := FALSE);
					usiStep				:= 0;
					usiCount			:= 0;
					bNotInterruptible	:= FALSE;
					tyParamOutDriver.uiCtrlword_6040.7	:= FALSE;
					sStatTxt	:= a_sStatText[eStat];

				END_IF

				eStatus	:= Idle;

				IF EDGENEG(p_bManual) THEN
					fMotionCANRstCtrlWord(ADR(tyParamOutDriver));
				END_IF

			PPActGoWidth:
				IF (eStatus = Idle OR eStatus = Busy) THEN

					eStatus	:= Busy;

					sStatTxt	:= a_sStatText[eStat];

					bNotInterruptible	:= TRUE;

					CASE usiStep OF
						0:	//Wait For Motion Parameter Update
							p_diMovePosInUM	:= fAWWidthToPosInUM(p_diGoWidth , p_diWidthAtHmPos);
							usiStep	:= 1;

						1:	//Check Position Difference
							IF tyParamOut.bPosDiff = TRUE THEN
								usiStep	:= 2;
							ELSE
								eStatus	:= Done;
							END_IF

						2:	//Move
							fbFullMovAbsBl.tyParamInDriver					:= tyParamInDriver;
							fbFullMovAbsBl.tyParamInMove.diPosInUM			:= p_diMovePosInUM;
							fbFullMovAbsBl.tyParamInMove.diDistInUM			:= p_diMoveDistInUM;
							fbFullMovAbsBl.tyParamInMove.diVelInUMPS		:= p_diMoveVelInUMPS;
							fbFullMovAbsBl.tyParamInMove.diAcc				:= p_diMoveAcc;
							fbFullMovAbsBl.tyParamInMove.diDec				:= p_diMoveDec;
							fbFullMovAbsBl.tyParamOut						:= tyParamOut;
							fbFullMovAbsBl(bEn := TRUE);

							IF fbFullMovAbsBl.udiStatus = 0 THEN
								eStatus	:= Done;
							ELSIF fbFullMovAbsBl.udiStatus < 65534 THEN
								eStatus		:= Error;

								IF fbFullMovAbsBl.udiStatus = 1401 THEN
									udiStatus	:= 10002;	//Power On Time Out While Going New Width
								ELSIF fbFullMovAbsBl.udiStatus = 1402 THEN
									udiStatus	:= 10003;	//Homing Time Out While Going New Width
								ELSIF fbFullMovAbsBl.udiStatus = 1403 THEN
									udiStatus	:= 10004;	//Move Absolute Time Out While Going New Width
								ELSIF fbFullMovAbsBl.udiStatus = 1405 THEN
									udiStatus	:= 10005;	//Stop Motion Time Out While Going New Width
								ELSIF fbFullMovAbsBl.udiStatus = 1408 THEN
									udiStatus	:= 10006;	//Axis Error Reset Failed While Going New Width
								ELSIF fbFullMovAbsBl.udiStatus = 1409 THEN
									udiStatus	:= 10007;	//Axis Error Occur In Move Absolute While Going New Width
								ELSIF fbFullMovAbsBl.udiStatus = 1411 THEN
									udiStatus	:= 10008;	//Axis Error Occur In Homing While Going New Width
								ELSIF fbFullMovAbsBl.udiStatus = 1412 THEN
									udiStatus	:= 10009;	//Homing Done But Home Flag Is Not Activated While Going New Width
								ELSIF fbFullMovAbsBl.udiStatus = 1413 THEN
									udiStatus	:= 10010;	//Forward Limit Activated In Homing While Going New Width
								ELSIF fbFullMovAbsBl.udiStatus = 1414 THEN
									udiStatus	:= 10011;	//Reverse Limit Activated In Homing While Going New Width
								ELSIF fbFullMovAbsBl.udiStatus = 1415 THEN
									udiStatus	:= 10012;	//Forward Limit Activated In Move Absolute While Going New Width
								ELSIF fbFullMovAbsBl.udiStatus = 1416 THEN
									udiStatus	:= 10013;	//Reverse Limit Activated In Move Absolute While Going New Width
								ELSE
									udiStatus	:= fbFullMovAbsBl.udiStatus;
								END_IF
							END_IF

					END_CASE

				END_IF

			PPActGoWidthOff:
				IF (eStatus = Idle OR eStatus = Busy) THEN

					eStatus	:= Busy;

					sStatTxt	:= a_sStatText[eStat];

					bNotInterruptible	:= TRUE;

					CASE usiStep OF
						0:	//Wait For Motion Parameter Update
							p_diMovePosInUM	:= fAWWidthToPosInUM(p_diGoWidth , p_diWidthAtHmPos);
							usiStep	:= 1;

						1:	//Check Position Difference
							IF tyParamOut.bPosDiff = TRUE THEN
								usiStep	:= 2;
							ELSE
								eStatus	:= Done;
							END_IF

						2:	//Move
							fbFullMovAbsBl.tyParamInDriver					:= tyParamInDriver;
							fbFullMovAbsBl.tyParamInMove.diPosInUM			:= p_diMovePosInUM;
							fbFullMovAbsBl.tyParamInMove.diDistInUM			:= p_diMoveDistInUM;
							fbFullMovAbsBl.tyParamInMove.diVelInUMPS		:= p_diMoveVelInUMPS;
							fbFullMovAbsBl.tyParamInMove.diAcc				:= p_diMoveAcc;
							fbFullMovAbsBl.tyParamInMove.diDec				:= p_diMoveDec;
							fbFullMovAbsBl.tyParamOut						:= tyParamOut;
							fbFullMovAbsBl(bEn := TRUE);

							IF fbFullMovAbsBl.udiStatus = 0 THEN
								usiStep	:= 3;
							ELSIF fbFullMovAbsBl.udiStatus < 65534 THEN
								eStatus		:= Error;

								IF fbFullMovAbsBl.udiStatus = 1401 THEN
									udiStatus	:= 10035;	//Power On Time Out While Going New Width And Off
								ELSIF fbFullMovAbsBl.udiStatus = 1402 THEN
									udiStatus	:= 10036;	//Homing Time Out While Going New Width And Off
								ELSIF fbFullMovAbsBl.udiStatus = 1403 THEN
									udiStatus	:= 10037;	//Move Absolute Time Out While Going New Width And Off
								ELSIF fbFullMovAbsBl.udiStatus = 1405 THEN
									udiStatus	:= 10038;	//Stop Motion Time Out While Going New Width And Off
								ELSIF fbFullMovAbsBl.udiStatus = 1408 THEN
									udiStatus	:= 10039;	//Axis Error Reset Failed While Going New Width And Off
								ELSIF fbFullMovAbsBl.udiStatus = 1409 THEN
									udiStatus	:= 10040;	//Axis Error Occur In Move Absolute While Going New Width And Off
								ELSIF fbFullMovAbsBl.udiStatus = 1411 THEN
									udiStatus	:= 10041;	//Axis Error Occur In Homing While Going New Width And Off
								ELSIF fbFullMovAbsBl.udiStatus = 1412 THEN
									udiStatus	:= 10042;	//Homing Done But Home Flag Is Not Activated While Going New Width And Off
								ELSIF fbFullMovAbsBl.udiStatus = 1413 THEN
									udiStatus	:= 10043;	//Forward Limit Activated In Homing While Going New Width And Off
								ELSIF fbFullMovAbsBl.udiStatus = 1414 THEN
									udiStatus	:= 10044;	//Reverse Limit Activated In Homing While Going New Width And Off
								ELSIF fbFullMovAbsBl.udiStatus = 1415 THEN
									udiStatus	:= 10045;	//Forward Limit Activated In Move Absolute While Going New Width And Off
								ELSIF fbFullMovAbsBl.udiStatus = 1416 THEN
									udiStatus	:= 10046;	//Reverse Limit Activated In Move Absolute While Going New Width And Off
								ELSE
									udiStatus	:= fbFullMovAbsBl.udiStatus;
								END_IF
							END_IF

						3:	//Turn Off Motor
							fMotionCANRstCtrlWord(ADR(tyParamOutDriver));
							eStatus	:= Done;

					END_CASE

				END_IF

			PPActFullHm:
				IF (eStatus = Idle OR eStatus = Busy) THEN

					eStatus	:= Busy;

					sStatTxt	:= a_sStatText[eStat];

					bNotInterruptible	:= TRUE;

					fbFullHm.tyParamInDriver	:= tyParamInDriver;
					fbFullHm.tyParamOut			:= tyParamOut;
					fbFullHm(bEn := TRUE);

					IF fbFullHm.udiStatus = 0 THEN
						eStatus	:= Done;
					ELSIF fbFullHm.udiStatus < 65534 THEN
						eStatus		:= Error;

						IF fbFullHm.udiStatus = 1401 THEN
							udiStatus	:= 10014;	//Power On Time Out While Full Homing
						ELSIF fbFullHm.udiStatus = 1402 THEN
							udiStatus	:= 10015;	//Homing Time Out While Full Homing
						ELSIF fbFullHm.udiStatus = 1405 THEN
							udiStatus	:= 10016;	//Stop Motion Time Out While Full Homing
						ELSIF fbFullHm.udiStatus = 1408 THEN
							udiStatus	:= 10017;	//Axis Error Reset Failed While Full Homing
						ELSIF fbFullHm.udiStatus = 1411 THEN
							udiStatus	:= 10018;	//Axis Error Occur In Homing While Full Homing
						ELSIF fbFullHm.udiStatus = 1412 THEN
							udiStatus	:= 10019;	//Homing Done But Home Flag Is Not Activated While Full Homing
						ELSIF fbFullHm.udiStatus = 1413 THEN
							udiStatus	:= 10020;	//Forward Limit Activated In Homing While Full Homing
						ELSIF fbFullHm.udiStatus = 1414 THEN
							udiStatus	:= 10021;	//Reverse Limit Activated In Homing While Full Homing
						ELSE
							udiStatus	:= fbFullHm.udiStatus;
						END_IF
					END_IF

				END_IF

			PPActPwrOn:
				IF (eStatus = Idle OR eStatus = Busy) THEN

					eStatus	:= Busy;

					sStatTxt	:= a_sStatText[eStat];

					fbPwrOn.tyParamInDriver	:= tyParamInDriver;
					fbPwrOn(bEn := TRUE);

					IF fbPwrOn.udiStatus = 0 THEN
						eStatus	:= Done;
					ELSIF fbPwrOn.udiStatus < 65534 THEN
						eStatus		:= Error;

						IF fbPwrOn.udiStatus = 1401 THEN
							udiStatus	:= 10022;	//Power On Time Out
						ELSE
							udiStatus	:= fbPwrOn.udiStatus;
						END_IF
					END_IF

				END_IF

			PPActPwrOff:
				IF (eStatus = Idle OR eStatus = Busy) THEN

					eStatus	:= Busy;

					sStatTxt	:= a_sStatText[eStat];

					fbPwrOff.tyParamInDriver	:= tyParamInDriver;
					fbPwrOff(bEn := TRUE);

					IF fbPwrOff.udiStatus = 0 THEN
						eStatus	:= Done;
					ELSIF fbPwrOff.udiStatus < 65534 THEN
						eStatus		:= Error;

						IF fbPwrOff.udiStatus = 1400 THEN
							udiStatus	:= 10023;	//Power Off Time Out
						ELSE
							udiStatus	:= fbPwrOff.udiStatus;
						END_IF
					END_IF

				END_IF

			PPActHoming:

				IF (eStatus = Idle OR eStatus = Busy) THEN

					eStatus	:= Busy;

					sStatTxt	:= a_sStatText[eStat];

					bNotInterruptible	:= TRUE;

					fbHoming.tyParamInDriver	:= tyParamInDriver;
					fbHoming.tyParamOut			:= tyParamOut;
					fbHoming(bEn := TRUE);

					IF fbHoming.udiStatus = 0 THEN
						eStatus	:= Done;
					ELSIF fbHoming.udiStatus < 65534 THEN
						eStatus		:= Error;

						IF fbHoming.udiStatus = 1402 THEN
							udiStatus	:= 10024;	//Homing Time Out
						ELSIF fbHoming.udiStatus = 1411 THEN
							udiStatus	:= 10018;	//Axis Error Occur In Homing While Full Homing

						ELSIF fbHoming.udiStatus = 1413 THEN
							udiStatus	:= 10020;	//Forward Limit Activated In Homing While Full Homing
						ELSIF fbHoming.udiStatus = 1414 THEN
							udiStatus	:= 10021;	//Reverse Limit Activated In Homing While Full Homing
						ELSE
							udiStatus	:= fbHoming.udiStatus;
						END_IF
					END_IF

				END_IF

			PPActMovAbs:
				IF (eStatus = Idle OR eStatus = Busy) THEN

					eStatus	:= Busy;

					sStatTxt	:= a_sStatText[eStat];

					bNotInterruptible	:= TRUE;

					fbMovAbs.tyParamInDriver			:= tyParamInDriver;
					fbMovAbs.tyParamInMove.diPosInUM	:= p_diMovePosInUM;
					fbMovAbs.tyParamInMove.diDistInUM	:= p_diMoveDistInUM;
					fbMovAbs.tyParamInMove.diVelInUMPS	:= p_diMoveVelInUMPS;
					fbMovAbs.tyParamInMove.diAcc		:= p_diMoveAcc;
					fbMovAbs.tyParamInMove.diDec		:= p_diMoveDec;
					fbMovAbs(bEn := TRUE);

					IF fbMovAbs.udiStatus = 0 THEN
						eStatus	:= Done;
					ELSIF fbMovAbs.udiStatus < 65534 THEN
						eStatus		:= Error;

						IF fbMovAbs.udiStatus = 1403 THEN
							udiStatus	:= 10025;	//Move Absolute Time Out
						ELSE
							udiStatus	:= fbMovAbs.udiStatus;
						END_IF
					END_IF

				END_IF

			PPActMovRel:
				IF (eStatus = Idle OR eStatus = Busy) THEN

					eStatus	:= Busy;

					sStatTxt	:= a_sStatText[eStat];

					bNotInterruptible	:= TRUE;

					fbMovRel.tyParamInDriver			:= tyParamInDriver;
					fbMovRel.tyParamInMove.diPosInUM	:= p_diMovePosInUM;
					fbMovRel.tyParamInMove.diDistInUM	:= p_diMoveDistInUM;
					fbMovRel.tyParamInMove.diVelInUMPS	:= p_diMoveVelInUMPS;
					fbMovRel.tyParamInMove.diAcc		:= p_diMoveAcc;
					fbMovRel.tyParamInMove.diDec		:= p_diMoveDec;
					fbMovRel(bEn := TRUE);

					IF fbMovRel.udiStatus = 0 THEN
						eStatus	:= Done;
					ELSIF fbMovRel.udiStatus < 65534 THEN
						eStatus		:= Error;

						IF fbMovRel.udiStatus = 1404 THEN
							udiStatus	:= 10026;	//Move Relative Time Out
						ELSE
							udiStatus	:= fbMovRel.udiStatus;
						END_IF
					END_IF

				END_IF

			PPActJogOpen:
				IF (eStatus = Idle OR eStatus = Busy) THEN

					eStatus	:= Busy;

					sStatTxt	:= a_sStatText[eStat];

					bNotInterruptible	:= TRUE;

					fbJog.tyParamInDriver	:= tyParamInDriver;
					fbJog.tyParamInMove.diAcc		:= p_diMoveAcc;
					fbJog.tyParamInMove.diDec		:= p_diMoveDec;

					IF p_bDir = TRUE THEN
						fbJog.tyParamInJog.diVelInUMPS	:= p_diJogVelInUMPS;
					ELSE
						fbJog.tyParamInJog.diVelInUMPS	:= p_diJogVelInUMPS * -1;
					END_IF

					fbJog(bEn := TRUE);

					IF fbJog.udiStatus = 0 THEN
						bJogging	:= TRUE;
						bJogOpen	:= TRUE;
						eStatus		:= Done;
					ELSIF fbJog.udiStatus < 65534 THEN
						udiStatus	:= fbJog.udiStatus;
						eStatus		:= Error;
					END_IF

				END_IF

			PPActJogClose:
				IF (eStatus = Idle OR eStatus = Busy) THEN

					eStatus	:= Busy;

					sStatTxt	:= a_sStatText[eStat];

					bNotInterruptible	:= TRUE;

					fbJog.tyParamInDriver			:= tyParamInDriver;
					fbJog.tyParamInMove.diAcc		:= p_diMoveAcc;
					fbJog.tyParamInMove.diDec		:= p_diMoveDec;

					IF p_bDir = TRUE THEN
						fbJog.tyParamInJog.diVelInUMPS	:= p_diJogVelInUMPS * -1;
					ELSE
						fbJog.tyParamInJog.diVelInUMPS	:= p_diJogVelInUMPS;
					END_IF

					fbJog(bEn := TRUE);

					IF fbJog.udiStatus = 0 THEN
						bJogging	:= TRUE;
						bJogClose	:= TRUE;
						eStatus		:= Done;
					ELSIF fbJog.udiStatus < 65534 THEN
						udiStatus	:= fbJog.udiStatus;
						eStatus		:= Error;
					END_IF

				END_IF

			PPActJogStop:
				IF (eStatus = Idle OR eStatus = Busy) THEN

					sStatTxt	:= a_sStatText[eStat];

					fMotionCANJogStop(ADR(tyParamOutDriver));
					bJogging	:= FALSE;
					bJogClose	:= FALSE;
					bJogOpen	:= FALSE;
					eStatus	:= Done;

				END_IF

			PPActRstAxisErr:
				IF (eStatus = Idle OR eStatus = Busy) THEN

					eStatus	:= Busy;

					sStatTxt	:= a_sStatText[eStat];

					fbRstAxisErr(bEn := TRUE);

					IF fbRstAxisErr.udiStatus = 0 THEN
						eStatus	:= Done;
					ELSIF fbRstAxisErr.udiStatus < 65534 THEN
						udiStatus	:= fbRstAxisErr.udiStatus;
						eStatus		:= Error;
					END_IF

				END_IF

			PPActStop:
				IF (eStatus = Idle OR eStatus = Busy) THEN

					eStatus	:= Busy;

					sStatTxt	:= a_sStatText[eStat];

					fbStop.tyParamInDriver	:= tyParamInDriver;
					fbStop(bEn := TRUE);

					IF fbStop.udiStatus = 0 THEN
						bJogging	:= FALSE;
						bJogClose	:= FALSE;
						bJogOpen	:= FALSE;
						eStatus		:= Done;
					ELSIF fbStop.udiStatus < 65534 THEN
						eStatus		:= Error;

						IF fbStop.udiStatus = 1405 THEN
							udiStatus	:= 10027;	//Stop Motion Time Out
						ELSE
							udiStatus	:= fbStop.udiStatus;
						END_IF
					END_IF

				END_IF
		END_CASE

ELSE
	CASE eStat OF
		PPActSDOWrite:
			IF (eStatus = Idle OR eStatus = Busy) THEN

				eStatus	:= Busy;

				sStatTxt	:= a_sStatText[eStat];

				fbTm(IN := TRUE);

				IF fbTm.Q THEN

					fbSDOWrite.tyParamOut	:= tyParamOut;
					fbSDOWrite.tyTuning		:= p_tyTuning;

					fbSDOWrite(bEn := TRUE);

					IF fbSDOWrite.udiStatus = 0 THEN
						eStatus	:= Done;
					ELSIF fbSDOWrite.udiStatus < 65534 THEN
						fMotionCANRstCtrlWord(ADR(tyParamOutDriver));

						IF usiCount < 5 THEN
							fbTm(IN := FALSE);
							fbSDOWrite(bEn := FALSE);

							usiCount	:= usiCount + 1;
						ELSE
							eStatus	:= Error;

							IF fbSDOWrite.udiStatus = 1406 THEN
								udiStatus	:= 10028;	//SDO Write Error
							ELSE
								udiStatus	:= fbSDOWrite.udiStatus;
							END_IF
						END_IF

					END_IF

				END_IF

			END_IF

		PPActBGStartModOKChk:
			IF (eStatus = Idle OR eStatus = Busy) THEN

				sStatTxt	:= a_sStatText[eStat];

				bModuleOKChk	:= TRUE;
				eStatus			:= Done;

			END_IF

		PPActBGStopModOKChk:
			IF (eStatus = Idle OR eStatus = Busy) THEN

				sStatTxt	:= a_sStatText[eStat];

				bModuleOKChk	:= FALSE;
				eStatus			:= Done;

			END_IF

		PPActIdle:
			IF eStatus <> Idle THEN	//Reset Data
				//Private
				fbStop(bEn := FALSE);
				fbRstAxisErr(bEn := FALSE);
				fbJog(bEn := FALSE);
				fbMovRel(bEn := FALSE);
				fbMovAbs(bEn := FALSE);
				fbHoming(bEn := FALSE);
				fbPwrOff(bEn := FALSE);
				fbPwrOn(bEn := FALSE);
				fbFullHm(bEn := FALSE);
				fbFullMovAbs(bEn := FALSE);
				fbFullMovAbsBl(bEn := FALSE);
				fbSDOWrite(bEn := FALSE);
				fbTm(IN := FALSE);
				usiStep				:= 0;
				usiCount			:= 0;
				bNotInterruptible	:= FALSE;
				tyParamOutDriver.uiCtrlword_6040.7	:= FALSE;

				sStatTxt	:= a_sStatText[eStat];

			END_IF

			eStatus	:= Idle;

			IF EDGENEG(p_bManual) THEN
				fMotionCANRstCtrlWord(ADR(tyParamOutDriver));
			END_IF

		PPActRstNode:
			IF (eStatus = Idle OR eStatus = Busy) THEN

				eStatus	:= Busy;

				sStatTxt	:= a_sStatText[eStat];
				IF bRstErr THEN
					fbModuleOK(bEn := FALSE, bModuleOK := bModuleOK);
				END_IF
				fbModuleOK(bEn := TRUE);
				IF fbModuleOK.udiStatus = 0 THEN
					fbModuleOK(bEn := FALSE);
					eStatus			:= Done;
				ELSIF fbModuleOK.udiStatus < 65534 THEN
					eStatus		:= Error;

					IF fbModuleOK.udiStatus = 1407 THEN
						udiStatus	:= 10001;	//CANOpen Communication Error, ModuleOK Not TRUE
						fbModuleOK(bEn := FALSE);
					ELSE
						udiStatus	:= fbModuleOK.udiStatus;
					END_IF
				END_IF
			END_IF

		PPActRstAxisErr:
			IF (eStatus = Idle OR eStatus = Busy) THEN

				eStatus	:= Busy;

				sStatTxt	:= a_sStatText[eStat];

				fbRstAxisErr(bEn := TRUE);

				IF fbRstAxisErr.udiStatus = 0 THEN
					eStatus	:= Done;
				ELSIF fbRstAxisErr.udiStatus < 65534 THEN
					udiStatus	:= fbRstAxisErr.udiStatus;
					eStatus		:= Error;
				END_IF

			END_IF

	END_CASE
END_IF

END_ACTION
```

#### Act_RstErr.st
```iecst
(** 2020-03-16 **)
ACTION Act_RstErr:

	IF p_udiRstErr <> udiRstErrOld THEN
		bRstErr			:= TRUE;
		udiRstErrOld	:= p_udiRstErr;
		tyParamOutDriver.diJogVel_60FF	:= 0;
		bRstAndExt 		:= TRUE;

	ELSE
		bRstErr			:= FALSE;
	END_IF

	tyParamOutDriver.uiCtrlword_6040.7	:= bRstErr;

END_ACTION
```

#### Init.st
```iecst
(** 2019-04-24 **)
PROGRAM _INIT

	(* Always Change If Project Change *)

	//Pass Address To Global Address For External Use
	//Action, State & Status
	p_PPStat	:= ADR(eStat);
	p_PPStatus	:= ADR(eMainStatus);
	p_PPStatTxt	:= ADR(sStatTxt);

	//Alarm
	p_PPAlmData		:= ADR(tyAlmData);
	p_PPAlmData1	:= ADR(tyAlmData1);
	p_PPAlmData2	:= ADR(tyAlmData2);
	p_PPAlmData3	:= ADR(tyAlmData3);

	//Output
	p_PPParamOut		:= ADR(tyParamOut);
	p_PPPwrOn			:= ADR(tyParamOut.bPwrOn);
	p_PPIsHomed			:= ADR(tyParamOut.bIsHomed);
	p_PPPosDiff			:= ADR(tyParamOut.bPosDiff);
	p_PPAxisErr			:= ADR(tyParamOut.bAxisErr);
	p_PPAxisErrID		:= ADR(tyParamOut.udiAxisErrID);
	p_PPFwdLmtSen		:= ADR(tyParamOut.bFwdLmtSen);
	p_PPRevLmtSen		:= ADR(tyParamOut.bRevLmtSen);
	p_PPActualPos		:= ADR(tyParamOut.diActualPosInUM);
	p_PPAxisErrTxt		:= ADR(sAxisErrTxt);
	p_PPWidthPosDiff	:= ADR(bWidthPosDiff);
	p_PPJogging			:= ADR(bJogging);
	p_PPExtSen			:= ADR(bOpenSen);
	p_PPRetSen			:= ADR(bCloseSen);
	p_PPTurnToHm		:= ADR(bTurnToHm);
	(* Always Change If Project Change *)

END_PROGRAM
```

### DInput.typ
```iecst
(*2018-12-10*)
(**)
(*Data*)

TYPE
	tyDigitalInput : 	STRUCT
		bSafetyRlySig : BOOL;
		bEStopSig : BOOL;
		bCoverSWSig : BOOL;
		bDSBA : BOOL;
		bDSBB : BOOL;
		bPullerExtRS : BOOL;
		bPullerRetRS : BOOL;
		bPullerRotHmRS : BOOL;
		bPullerRotRmRS : BOOL;
		bConvLftSen : BOOL;
		bConvRgtSen : BOOL;
		bLifterTimingBeltSen : BOOL;
		bLifterSafetyLmtSW1 : BOOL;
		bLifterSafetyLmtSW2 : BOOL;
		bMag1FixedClampRS : BOOL;
		bMag1FixedUnclampRS : BOOL;
		bMag1RemoteClampRS : BOOL;
		bMag1RemoteUnclampRS : BOOL;
		bMag2FixedClampRS : BOOL;
		bMag2FixedUnclampRS : BOOL;
		bMag2RemoteClampRS : BOOL;
		bMag2RemoteUnclampRS : BOOL;
		bMag3FixedClampRS : BOOL;
		bMag3FixedUnclampRS : BOOL;
		bMag3RemoteClampRS : BOOL;
		bMag3RemoteUnclampRS : BOOL;
		bMag4FixedClampRS : BOOL;
		bMag4FixedUnclampRS : BOOL;
		bMag4RemoteClampRS : BOOL;
		bMag4RemoteUnclampRS : BOOL;
		bInShutterOpenRS : BOOL;
		bInShutterCloseRS : BOOL;
		bOutShutterOpenRS : BOOL;
		bOutShutterCloseRS : BOOL;
		bMagPresentSen1 : BOOL;
		bMagPresentSen2 : BOOL;
		bMagPresentSen3 : BOOL;
		bMagPresentSen4 : BOOL;
		bMagConvEntSen1 : BOOL;
		bMagConvEntSen2 : BOOL;
		bMagConvEntSen3 : BOOL;
		bMagConvEntSen4 : BOOL;
		bMag1AGVInPosSen1 : BOOL;
		bMag1AGVInPosSen2 : BOOL;
		bMag2AGVInPosSen1 : BOOL;
		bMag2AGVInPosSen2 : BOOL;
		bMag3AGVInPosSen1 : BOOL;
		bMag3AGVInPosSen2 : BOOL;
		bMag4AGVInPosSen1 : BOOL;
		bMag4AGVInPosSen2 : BOOL;
		bMag1OrientChkSen1 : BOOL;
		bMag1OrientChkSen2 : BOOL;
		bMag2OrientChkSen1 : BOOL;
		bMag2OrientChkSen2 : BOOL;
		bMag3OrientChkSen1 : BOOL;
		bMag3OrientChkSen2 : BOOL;
		bMag4OrientChkSen1 : BOOL;
		bMag4OrientChkSen2 : BOOL;
		bDSWidthChkSen : BOOL;
		bMagConvHeightSen1 : BOOL;
		bMagConvHeightSen2 : BOOL;
		bMagConvHeightSen3 : BOOL;
		bMagConvHeightSen4 : BOOL;
		bMagConvSmallMagSen1 : BOOL;
		bMagConvSmallMagSen2 : BOOL;
		bMagConvSmallMagSen3 : BOOL;
		bMagConvSmallMagSen4 : BOOL;
		bMagConvLargeMagSen1 : BOOL;
		bMagConvLargeMagSen2 : BOOL;
		bMagConvLargeMagSen3 : BOOL;
		bMagConvLargeMagSen4 : BOOL;
		bMagConvCAB717MagSen1 : BOOL;
		bMagConvCAB717MagSen2 : BOOL;
		bMagConvCAB717MagSen3 : BOOL;
		bMagConvCAB717MagSen4 : BOOL;
		bMag1SelUnClampRS : BOOL;
		bMag2SelUnClampRS : BOOL;
		bMag3SelUnClampRS : BOOL;
		bMag4SelUnClampRS : BOOL;
		bSOT1Receive : BOOL;
		bSOT1AIVError : BOOL;
		bSOT1AIVSizeLarge : BOOL;
		bSOT1AIVReady : BOOL;
		bSOT1AIVAvailable : BOOL;
		bSOT2Receive : BOOL;
		bSOT2AIVError : BOOL;
		bSOT2AIVSizeLarge : BOOL;
		bSOT2AIVReady : BOOL;
		bSOT2AIVAvailable : BOOL;
		bSOT3Receive : BOOL;
		bSOT3AIVError : BOOL;
		bSOT3AIVSizeLarge : BOOL;
		bSOT3AIVReady : BOOL;
		bSOT3AIVAvailable : BOOL;
		bSOT4Receive : BOOL;
		bSOT4AIVError : BOOL;
		bSOT4AIVSizeLarge : BOOL;
		bSOT4AIVReady : BOOL;
		bSOT4AIVAvailable : BOOL;
		bFleetManagerReady : BOOL;
		bPullerExtSlwSen : BOOL;
		bPullerRetSlwSen : BOOL;
		bMtrPullerTorqueSig : BOOL;
		bMtrPullerAlmSig : BOOL;
		bMag1SafetyBarExtRS : BOOL;
		bMag1SafetyBarRetRS : BOOL;
		bMag2SafetyBarExtRS : BOOL;
		bMag2SafetyBarRetRS : BOOL;
		bMag3SafetyBarExtRS : BOOL;
		bMag3SafetyBarRetRS : BOOL;
		bMag4SafetyBarExtRS : BOOL;
		bMag4SafetyBarRetRS : BOOL;
		bMagWidthChkSen : BOOL;
		bPullerAntiJam : BOOL;
		bCurtainSensor : BOOL;
		bBypCurtainSensorPB : BOOL;
		bInShutterOpenRS2 : BOOL;
		bInShutterCloseRS2 : BOOL;
		bInShutterOpenRS3 : BOOL;
		bInShutterCloseRS3 : BOOL;
		bMag1FixedSideDetect : BOOL;
		bMag1RemoteSideDetect : BOOL;
		bMag2FixedSideDetect : BOOL;
		bMag2RemoteSideDetect : BOOL;
		bMag3FixedSideDetect : BOOL;
		bMag3RemoteSideDetect : BOOL;
		bCurtainSafetySig2 : BOOL;
		bHighMagDetSen1 : BOOL;
		bHighMagDetSen2 : BOOL;
		bHighMagDetSen3 : BOOL;
		bConvClrSen : BOOL;
		bDSSafetySig : BOOL;
		bDSUnlockCoverSig : BOOL;
		bOutShutterOpenRS2 : BOOL;
		bOutShutterCloseRS2 : BOOL;
		bTrolleyExtRS1 : BOOL;
		bTrolleyExtRS2 : BOOL;
		bTrolleyPreSen1 : BOOL;
		bTrolleyPreSen2 : BOOL;
		bSlotLckSenMag1 : BOOL;
		bSlotLckSenMag2 : BOOL;
		bSPARE16 : BOOL;
		bSPARE17 : BOOL;
		bSPARE18 : BOOL;
		bSPARE19 : BOOL;
		bSPARE20 : BOOL;
	END_STRUCT;
	tyDigitalInputSettings : 	STRUCT
		diSafetyRlySig : DINT;
		diEStopSig : DINT;
		diCoverSWSig : DINT;
		diDSBA : DINT;
		diDSBB : DINT;
		diPullerExtRS : DINT;
		diPullerRetRS : DINT;
		diPullerRotHmRS : DINT;
		diPullerRotRmRS : DINT;
		diConvLftSen : DINT;
		diConvRgtSen : DINT;
		diLifterTimingBeltSen : DINT;
		diLifterSafetyLmtSW1 : DINT;
		diLifterSafetyLmtSW2 : DINT;
		diMag1FixedClampRS : DINT;
		diMag1FixedUnclampRS : DINT;
		diMag1RemoteClampRS : DINT;
		diMag1RemoteUnclampRS : DINT;
		diMag2FixedClampRS : DINT;
		diMag2FixedUnclampRS : DINT;
		diMag2RemoteClampRS : DINT;
		diMag2RemoteUnclampRS : DINT;
		diMag3FixedClampRS : DINT;
		diMag3FixedUnclampRS : DINT;
		diMag3RemoteClampRS : DINT;
		diMag3RemoteUnclampRS : DINT;
		diMag4FixedClampRS : DINT;
		diMag4FixedUnclampRS : DINT;
		diMag4RemoteClampRS : DINT;
		diMag4RemoteUnclampRS : DINT;
		diInShutterOpenRS : DINT;
		diInShutterCloseRS : DINT;
		diOutShutterOpenRS : DINT;
		diOutShutterCloseRS : DINT;
		diMagPresentSen1 : DINT;
		diMagPresentSen2 : DINT;
		diMagPresentSen3 : DINT;
		diMagPresentSen4 : DINT;
		diMagConvEntSen1 : DINT;
		diMagConvEntSen2 : DINT;
		diMagConvEntSen3 : DINT;
		diMagConvEntSen4 : DINT;
		diMag1AGVInPosSen1 : DINT;
		diMag1AGVInPosSen2 : DINT;
		diMag2AGVInPosSen1 : DINT;
		diMag2AGVInPosSen2 : DINT;
		diMag3AGVInPosSen1 : DINT;
		diMag3AGVInPosSen2 : DINT;
		diMag4AGVInPosSen1 : DINT;
		diMag4AGVInPosSen2 : DINT;
		diMag1OrientChkSen1 : DINT;
		diMag1OrientChkSen2 : DINT;
		diMag2OrientChkSen1 : DINT;
		diMag2OrientChkSen2 : DINT;
		diMag3OrientChkSen1 : DINT;
		diMag3OrientChkSen2 : DINT;
		diMag4OrientChkSen1 : DINT;
		diMag4OrientChkSen2 : DINT;
		diDSWidthChkSen : DINT;
		diMagConvHeightSen1 : DINT;
		diMagConvHeightSen2 : DINT;
		diMagConvHeightSen3 : DINT;
		diMagConvHeightSen4 : DINT;
		diMagConvSmallMagSen1 : DINT;
		diMagConvSmallMagSen2 : DINT;
		diMagConvSmallMagSen3 : DINT;
		diMagConvSmallMagSen4 : DINT;
		diMagConvLargeMagSen1 : DINT;
		diMagConvLargeMagSen2 : DINT;
		diMagConvLargeMagSen3 : DINT;
		diMagConvLargeMagSen4 : DINT;
		diMagConvCAB717MagSen1 : DINT;
		diMagConvCAB717MagSen2 : DINT;
		diMagConvCAB717MagSen3 : DINT;
		diMagConvCAB717MagSen4 : DINT;
		diMag1SelUnClampRS : DINT;
		diMag2SelUnClampRS : DINT;
		diMag3SelUnClampRS : DINT;
		diMag4SelUnClampRS : DINT;
		diSOT1Receive : DINT;
		diSOT1AIVError : DINT;
		diSOT1AIVSizeLarge : DINT;
		diSOT1AIVReady : DINT;
		diSOT1AIVAvailable : DINT;
		diSOT2Receive : DINT;
		diSOT2AIVError : DINT;
		diSOT2AIVSizeLarge : DINT;
		diSOT2AIVReady : DINT;
		diSOT2AIVAvailable : DINT;
		diSOT3Receive : DINT;
		diSOT3AIVError : DINT;
		diSOT3AIVSizeLarge : DINT;
		diSOT3AIVReady : DINT;
		diSOT3AIVAvailable : DINT;
		diSOT4Receive : DINT;
		diSOT4AIVError : DINT;
		diSOT4AIVSizeLarge : DINT;
		diSOT4AIVReady : DINT;
		diSOT4AIVAvailable : DINT;
		diFleetManagerReady : DINT;
		diPullerExtSlwSen : DINT;
		diPullerRetSlwSen : DINT;
		diMtrPullerTorqueSig : DINT;
		diMtrPullerAlmSig : DINT;
		diMag1SafetyBarExtRS : DINT;
		diMag1SafetyBarRetRS : DINT;
		diMag2SafetyBarExtRS : DINT;
		diMag2SafetyBarRetRS : DINT;
		diMag3SafetyBarExtRS : DINT;
		diMag3SafetyBarRetRS : DINT;
		diMag4SafetyBarExtRS : DINT;
		diMag4SafetyBarRetRS : DINT;
		diMagWidthChkSen : DINT;
		diPullerAntiJam : DINT;
		diCurtainSensor : DINT;
		diBypCurtainSensorPB : DINT;
		diInShutterOpenRS2 : DINT;
		diInShutterCloseRS2 : DINT;
		diInShutterOpenRS3 : DINT;
		diInShutterCloseRS3 : DINT;
		diMag1FixedSideDetect : DINT;
		diMag1RemoteSideDetect : DINT;
		diMag2FixedSideDetect : DINT;
		diMag2RemoteSideDetect : DINT;
		diMag3FixedSideDetect : DINT;
		diMag3RemoteSideDetect : DINT;
		diCurtainSafetySig2 : DINT;
		diHighMagDetSen1 : DINT;
		diHighMagDetSen2 : DINT;
		diHighMagDetSen3 : DINT;
		diConvClrSen : DINT;
		diDSUnlockCoverSig : DINT;
		diDSSafetySig : DINT;
		diOutShutterOpenRS2 : DINT;
		diOutShutterCloseRS2 : DINT;
		diTrolleyExtRS1 : DINT;
		diTrolleyExtRS2 : DINT;
		diTrolleyPreSen1 : DINT;
		diTrolleyPreSen2 : DINT;
		diSlotLckSenMag1 : DINT;
		diSlotLckSenMag2 : DINT;
		diSPARE16 : DINT;
		diSPARE17 : DINT;
		diSPARE18 : DINT;
		diSPARE19 : DINT;
		diSPARE20 : DINT;
	END_STRUCT;
	tySOTSigmulateSig : 	STRUCT
		tyBtnInPos : BOOL;
		tyBtnError : BOOL;
		tyBtnRdy : BOOL;
		tyBtnAvail : BOOL;
	END_STRUCT;
END_TYPE
```

### DInput.var
```iecst
(*2018-12-10*)
(**)
(*Constant*)
VAR CONSTANT
	c_udiDInputMax : UDINT := 300; (*Constant Digital Input Quantity (+1 For Damaged) (+1 For Spare)*)
END_VAR
(**)
(*Action & State & Status*)
(**)
(*Alarm*)
VAR
	p_DIAlmData1 : UDINT;
	p_DIAlmData2 : UDINT;
	p_DIAlmData3 : UDINT;
	p_DIAlmData4 : UDINT;
	p_DIAlmData5 : UDINT;
	p_DIAlmData6 : UDINT;
END_VAR
(**)
(*Output*)
VAR
	p_DI : UDINT;
	p_DISafetyRlySig : UDINT;
	p_DIEStopSig : UDINT;
	p_DICoverSWSig : UDINT;
	p_DIDSBA : UDINT;
	p_DIDSBB : UDINT;
	p_DIPullerExtRS : UDINT;
	p_DIPullerRetRS : UDINT;
	p_DIPullerRotHmRS : UDINT;
	p_DIPullerRotRmRS : UDINT;
	p_DIConvLftSen : UDINT;
	p_DIConvRgtSen : UDINT;
	p_DILifterTimingBeltSen : UDINT;
	p_DILifterSafetyLmtSW1 : UDINT;
	p_DILifterSafetyLmtSW2 : UDINT;
	p_DIMag1FixedClampRS : UDINT;
	p_DIMag1FixedUnclampRS : UDINT;
	p_DIMag1RemoteClampRS : UDINT;
	p_DIMag1RemoteUnclampRS : UDINT;
	p_DIMag2FixedClampRS : UDINT;
	p_DIMag2FixedUnclampRS : UDINT;
	p_DIMag2RemoteClampRS : UDINT;
	p_DIMag2RemoteUnclampRS : UDINT;
	p_DIMag3FixedClampRS : UDINT;
	p_DIMag3FixedUnclampRS : UDINT;
	p_DIMag3RemoteClampRS : UDINT;
	p_DIMag3RemoteUnclampRS : UDINT;
	p_DIMag4FixedClampRS : UDINT;
	p_DIMag4FixedUnclampRS : UDINT;
	p_DIMag4RemoteClampRS : UDINT;
	p_DIMag4RemoteUnclampRS : UDINT;
	p_DIInShutterOpenRS : UDINT;
	p_DIInShutterCloseRS : UDINT;
	p_DIInShutterOpenRS2 : UDINT;
	p_DIInShutterCloseRS2 : UDINT;
	p_DIInShutterOpenRS3 : UDINT;
	p_DIInShutterCloseRS3 : UDINT;
	p_DIOutShutterOpenRS : UDINT;
	p_DIOutShutterCloseRS : UDINT;
	p_DIOutShutterOpenRS2 : UDINT;
	p_DIOutShutterCloseRS2 : UDINT;
	p_DIMagPresentSen1 : UDINT;
	p_DIMagPresentSen2 : UDINT;
	p_DIMagPresentSen3 : UDINT;
	p_DIMagPresentSen4 : UDINT;
	p_DIMagConvEntSen1 : UDINT;
	p_DIMagConvEntSen2 : UDINT;
	p_DIMagConvEntSen3 : UDINT;
	p_DIMagConvEntSen4 : UDINT;
	p_DIMag1AGVInPosSen1 : UDINT;
	p_DIMag1AGVInPosSen2 : UDINT;
	p_DIMag2AGVInPosSen1 : UDINT;
	p_DIMag2AGVInPosSen2 : UDINT;
	p_DIMag3AGVInPosSen1 : UDINT;
	p_DIMag3AGVInPosSen2 : UDINT;
	p_DIMag4AGVInPosSen1 : UDINT;
	p_DIMag4AGVInPosSen2 : UDINT;
	p_DIMag1OrientChkSen1 : UDINT;
	p_DIMag1OrientChkSen2 : UDINT;
	p_DIMag2OrientChkSen1 : UDINT;
	p_DIMag2OrientChkSen2 : UDINT;
	p_DIMag3OrientChkSen1 : UDINT;
	p_DIMag3OrientChkSen2 : UDINT;
	p_DIMag4OrientChkSen1 : UDINT;
	p_DIMag4OrientChkSen2 : UDINT;
	p_DIDSWidthChkSen : UDINT;
	p_DIMagConvHeightSen1 : UDINT;
	p_DIMagConvHeightSen2 : UDINT;
	p_DIMagConvHeightSen3 : UDINT;
	p_DIMagConvHeightSen4 : UDINT;
	p_DIMagConvSmallMagSen1 : UDINT;
	p_DIMagConvSmallMagSen2 : UDINT;
	p_DIMagConvSmallMagSen3 : UDINT;
	p_DIMagConvSmallMagSen4 : UDINT;
	p_DIMagConvLargeMagSen1 : UDINT;
	p_DIMagConvLargeMagSen2 : UDINT;
	p_DIMagConvLargeMagSen3 : UDINT;
	p_DIMagConvLargeMagSen4 : UDINT;
	p_DIMagConvCAB717MagSen1 : UDINT;
	p_DIMagConvCAB717MagSen2 : UDINT;
	p_DIMagConvCAB717MagSen3 : UDINT;
	p_DIMagConvCAB717MagSen4 : UDINT;
	p_DIMag1SelUnclampRS : UDINT;
	p_DIMag2SelUnclampRS : UDINT;
	p_DIMag3SelUnclampRS : UDINT;
	p_DIMag4SelUnclampRS : UDINT;
	p_DISOT1Receive : UDINT;
	p_DISOT1Error : UDINT;
	p_DISOT1SizeLarge : UDINT;
	p_DISOT1Ready : UDINT;
	p_DISOT1Available : UDINT;
	p_DISOT2Receive : UDINT;
	p_DISOT2Error : UDINT;
	p_DISOT2SizeLarge : UDINT;
	p_DISOT2Ready : UDINT;
	p_DISOT2Available : UDINT;
	p_DISOT3Receive : UDINT;
	p_DISOT3Error : UDINT;
	p_DISOT3SizeLarge : UDINT;
	p_DISOT3Ready : UDINT;
	p_DISOT3Available : UDINT;
	p_DISOT4Receive : UDINT;
	p_DISOT4Error : UDINT;
	p_DISOT4SizeLarge : UDINT;
	p_DISOT4Ready : UDINT;
	p_DISOT4Available : UDINT;
	p_DIFleetManagerActive : UDINT;
	p_DIPullerExtSlwSen : UDINT;
	p_DIPullerRetSlwSen : UDINT;
	p_DIMtrPullerTorqueSig : UDINT;
	p_DIMtrPullerAlmSig : UDINT;
	p_DIMag1SafetyBarExtRS : UDINT;
	p_DIMag1SafetyBarRetRS : UDINT;
	p_DIMag2SafetyBarExtRS : UDINT;
	p_DIMag2SafetyBarRetRS : UDINT;
	p_DIMag3SafetyBarExtRS : UDINT;
	p_DIMag3SafetyBarRetRS : UDINT;
	p_DIMag4SafetyBarExtRS : UDINT;
	p_DIMag4SafetyBarRetRS : UDINT;
	p_DIMagWidthChkSen : UDINT;
	p_DIMcSelfTest : UDINT;
	p_DISimServoEn : UDINT;
	p_DIPullerAntiJamSen : UDINT;
	p_DICurtainSen : UDINT;
	p_DIBypCurtainSensorPB : UDINT;
	p_DICurtainSafetySig2 : UDINT;
	p_DIMag1FixedSideDetect : UDINT;
	p_DIMag1RemoteSideDetect : UDINT;
	p_DIMag2FixedSideDetect : UDINT;
	p_DIMag2RemoteSideDetect : UDINT;
	p_DIMag3FixedSideDetect : UDINT;
	p_DIMag3RemoteSideDetect : UDINT;
	p_DIHighMagDetSen1 : UDINT;
	p_DIHighMagDetSen2 : UDINT;
	p_DIHighMagDetSen3 : UDINT;
	p_DIConvClrSen : UDINT;
	p_DIDSSafetySig : UDINT;
	p_DIDSUnlockSafetySig : UDINT;
	p_DITrolleyExtRS1 : UDINT;
	p_DITrolleyExtRS2 : UDINT;
	p_DITrolleyPreSen1 : UDINT;
	p_DITrolleyPreSen2 : UDINT;
	p_DISlotLckSenMag1 : UDINT;
	p_DISlotLckSenMag2 : UDINT;
END_VAR
```

### Program Logical/DInput/DInput

#### InputRef.var
```iecst
(*2019-03-22*)
(**)
(*General*)
VAR
	p_udiMax : REFERENCE TO UDINT;
	p_udiRstErr : REFERENCE TO UDINT;
END_VAR
(**)
(*Configuration*)
VAR
	p_tyDISettings : REFERENCE TO tyDigitalInputSettings;
	p_sProgNm : REFERENCE TO STRING[15];
END_VAR
(**)
VAR
	p_diConvLftSenOnTm : REFERENCE TO DINT;
	p_diConvLftSenOffTm : REFERENCE TO DINT;
	p_diConvRgtSenOnTm : REFERENCE TO DINT;
	p_diConvRgtSenOffTm : REFERENCE TO DINT;
	p_diMagConvEntSenOnTm : REFERENCE TO DINT;
	p_diMagConvEntSenOffTm : REFERENCE TO DINT;
	p_diMagConvPresentSenOnTm : REFERENCE TO DINT;
	p_diMagConvPresentSenOffTm : REFERENCE TO DINT;
	p_diConvClrSenOnTm : REFERENCE TO DINT;
	p_diConvClrSenOffTm : REFERENCE TO DINT;
	p_diTrolleySenOnTm : REFERENCE TO DINT;
	p_diTrolleySenOffTm : REFERENCE TO DINT;
	p_tySOTSimulate1 : REFERENCE TO tySOTSigmulateSig;
	p_tySOTSimulate2 : REFERENCE TO tySOTSigmulateSig;
	p_tySOTSimulate3 : REFERENCE TO tySOTSigmulateSig;
	p_tySOTSimulate4 : REFERENCE TO tySOTSigmulateSig;
	p_bUIAGVSimulationOn : REFERENCE TO BOOL;
	p_eAGVComProtocol : REFERENCE TO eMcAGVCommProtocol;
	p_tyTagFromMes : REFERENCE TO tyStatFromMES;
	p_tyDO : REFERENCE TO tyDigitalOutput;
	p_eLDMag : REFERENCE TO eLDMag;
	p_bPullConvHvBrd : REFERENCE TO BOOL;
	p_bRstErrSafetyRlyRst : REFERENCE TO BOOL;
	p_bRstCurtainSenCtrl : REFERENCE TO BOOL;
	p_bLinkStartupRun : REFERENCE TO BOOL;
END_VAR
```

#### InputRef_Link.var
```iecst
(*2019-04-09*)
(**)
(*External Data*)
VAR
	p_eLinkAGVComProtocol : REFERENCE TO eMcAGVCommProtocol;
	p_bLinkNtParamProjSOTSenPrep : REFERENCE TO BOOL;
	p_bOpsTravLifLDBypCurtainSenCtrl : REFERENCE TO BOOL;
	p_bCurtainSenPrep : REFERENCE TO BOOL;
END_VAR
```

#### Local.var
```iecst
(*2019-03-25*)
(**)
(*Local Action, State & Status*)
VAR
	eStatus1 : eFBStatus := Idle;
	eStatus2 : eFBStatus := Idle;
	eStatus3 : eFBStatus := Idle;
	eStatus4 : eFBStatus := Idle;
	eStatus5 : eFBStatus := Idle;
	eStatus6 : eFBStatus := Idle;
	udiStatus1 : UDINT := 0;
	udiStatus2 : UDINT := 0;
	udiStatus3 : UDINT := 0;
	udiStatus4 : UDINT := 0;
	udiStatus5 : UDINT := 0;
	udiStatus6 : UDINT := 0;
END_VAR
(**)
(*Local Alarm*)
VAR
	tyAlmData1 : tyAlmDat;
	tyAlmData2 : tyAlmDat;
	tyAlmData3 : tyAlmDat;
	tyAlmData4 : tyAlmDat;
	tyAlmData5 : tyAlmDat;
	tyAlmData6 : tyAlmDat;
	a_tyAlmText : ARRAY[10000..10099] OF tyAlmTxt := [(sAlmText:='Emergency Stop Button Pressed',sRcyText:='Release The Emergency Stop Button And Reset The Error To Resume Operation.'),(sAlmText:='Door / Cover Opened',sRcyText:='Close The Door / Cover Tightly And Resume Operation.'),(sAlmText:='Lifter Timing Belt Broken',sRcyText:='Replace New Lifter Timing Belt.'),(sAlmText:='Lifter Reached Safety Limit Switch',sRcyText:='Move Lifter Upward And Make Sure There Is No Obstable Interrupting Lifter.'),(sAlmText:='Safety Relay Signal Off',sRcyText:='Please Check The Safety Relay Signal'),(sAlmText:='Safety Curtain Sensor Activated',sRcyText:='Please Clear The Area Of Safety Curtain Sensor And Resume Operation.'),94(0)];
END_VAR
(**)
(*Local Output*)
VAR
	tyDInput : tyDigitalInput;
	bSimServoEn : BOOL := TRUE;
END_VAR
(**)
(*Local Input*)
VAR
	udiRstErr : UDINT := 0;
	tyDISettings : tyDigitalInputSettings := (0);
	sProgNm : STRING[15] := 'DInput';
END_VAR
(**)
VAR
	diConvLftSenOnTm : DINT := 0;
	diConvLftSenOffTm : DINT := 50;
	diConvRgtSenOnTm : DINT := 0;
	diConvRgtSenOffTm : DINT := 50;
	diMagConvEntSenOnTm : DINT := 0;
	diMagConvEntSenOffTm : DINT := 50;
	diMagConvPresentSenOnTm : DINT := 0;
	diMagConvPresentSenOffTm : DINT := 50;
	diConvClrSenOnTm : DINT := 0;
	diConvClrSenOffTm : DINT := 0;
	diTrolleySenOnTm : DINT := 1200;
	diTrolleySenOffTm : DINT := 0;
END_VAR
(**)
(*Local*)
VAR
	bRstErr : BOOL;
	udiRstErrOld : UDINT;
	bInitDone : BOOL;
	bInitialDone : BOOL;
	bSafetySigErrNoBuz : BOOL;
	a_bPhysicalDI : ARRAY[1..c_udiDInputMax] OF BOOL;
	fbConvLftSigFltr : fbSenFltr;
	fbConvRgtSigFltr : fbSenFltr;
	fbConvClrSigFltr : fbSenFltr;
	fbMagConv1EntSigFltr : fbSenFltr;
	fbMagConv2EntSigFltr : fbSenFltr;
	fbMagConv3EntSigFltr : fbSenFltr;
	fbMagConv4EntSigFltr : fbSenFltr;
	fbMagConv1PresentSigFltr : fbSenFltr;
	fbMagConv2PresentSigFltr : fbSenFltr;
	fbMagConv3PresentSigFltr : fbSenFltr;
	fbMagConv4PresentSigFltr : fbSenFltr;
	fbTrolley1PresentSigFltr : fbSenFltr;
	fbTrolley2PresentSigFltr : fbSenFltr;
	bAgvComIODisabled : BOOL;
	fbSelfTestTm1 : TON := (PT:=T#10s);
	fbSelfTestTm2 : TON := (PT:=T#10s);
	fbSelfTestTm3 : TON := (PT:=T#10s);
	fbSelfTestTm4 : TON := (PT:=T#10s);
	bSelfTest : BOOL := FALSE;
	fbConvLftSenTm : TON := (PT:=T#1s);
	fbSafetyRlyRstTm : TON := (PT:=T#2s);
	fbCurtainSafetyRstTm : TON := (PT:=T#200ms);
	udiModuleNum : UDINT := 5751;
END_VAR
```

#### Act_Alarm2.st
```iecst
(** 2019-03-25 **)
ACTION Act_Alarm2:

	//Error
	IF EDGEPOS(eStatus2 = Error) THEN

		tyAlmData2.sProgNm		:= p_sProgNm;
		tyAlmData2.udiCode		:= udiStatus2;
		tyAlmData2.eSeverity	:= AlmSeverityError;
		tyAlmData2.udiRunTime	:= tyAlmData2.udiRunTime + 1;
		tyAlmData2.bAlm			:= TRUE;
		tyAlmData2.udiModuleNum  := udiModuleNum;

		//Get Error Message
		IF tyAlmData2.udiCode < 10000 OR tyAlmData2.udiCode > 10099 THEN
			tyAlmData2.sAlmMsg	:= 'Unknown';
			tyAlmData2.sRcyMsg	:= 'Unknown';
		ELSE
			tyAlmData2.sAlmMsg	:= a_tyAlmText[tyAlmData2.udiCode].sAlmText;
			tyAlmData2.sRcyMsg	:= a_tyAlmText[tyAlmData2.udiCode].sRcyText;
		END_IF

	ELSIF bRstErr AND (tyAlmData2.udiCode <> 0) THEN

		tyAlmData2.udiCode		:= 0;
		tyAlmData2.eSeverity	:= AlmSeverityNA;
		tyAlmData2.sAlmMsg		:= '';
		tyAlmData2.sRcyMsg		:= '';
		tyAlmData2.bAlm			:= FALSE;
	END_IF

END_ACTION
```

#### Act_Alarm6.st
```iecst
(** Added By JOHN **)
ACTION Act_Alarm6:

	//Error
	IF EDGEPOS(eStatus6 = Error) THEN

		tyAlmData6.sProgNm		:= p_sProgNm;
		tyAlmData6.udiCode		:= udiStatus6;
		tyAlmData6.eSeverity	:= AlmSeverityError;
		tyAlmData6.udiRunTime	:= tyAlmData6.udiRunTime + 1;
		tyAlmData6.bAlm			:= TRUE;
		tyAlmData6.udiModuleNum  := udiModuleNum;
		g_sDInputProgNm		:= p_sProgNm;
		//Get Error Message
		IF tyAlmData6.udiCode < 10000 OR tyAlmData6.udiCode > 10099 THEN
			tyAlmData6.sAlmMsg	:= 'Unknown';
			tyAlmData6.sRcyMsg	:= 'Unknown';
		ELSE
			tyAlmData6.sAlmMsg	:= a_tyAlmText[tyAlmData6.udiCode].sAlmText;
			tyAlmData6.sRcyMsg	:= a_tyAlmText[tyAlmData6.udiCode].sRcyText;
		END_IF

	ELSIF bRstErr AND (tyAlmData6.udiCode <> 0) THEN

		tyAlmData6.udiCode		:= 0;
		tyAlmData6.eSeverity	:= AlmSeverityNA;
		tyAlmData6.sAlmMsg		:= '';
		tyAlmData6.sRcyMsg		:= '';
		tyAlmData6.bAlm			:= FALSE;
	END_IF

END_ACTION
```
